LIN {X 0,Y 303.752,Z 774.326,A -85,B 0,C 180,E1 -15927.348,E2 -15927.348} C_VEL
LIN {X 0,Y 303.832,Z 775.153,A -85,B 0,C 180,E1 -15928.675,E2 -15928.675} C_VEL
LIN {X 0,Y 303.933,Z 775.529,A -85,B 0,C 180,E1 -15930,E2 -15930} C_VEL
LIN {X 0,Y 303.82,Z 775.489,A -85,B 0,C 180,E1 -15931.325,E2 -15931.325} C_VEL
LIN {X 0,Y 303.73,Z 775.052,A -85,B 0,C 180,E1 -15932.652,E2 -15932.652} C_VEL
LIN {X 0,Y 303.716,Z 774.21,A -85,B 0,C 180,E1 -15933.981,E2 -15933.981} C_VEL
LIN {X 0,Y 303.694,Z 772.494,A -85,B 0,C 180,E1 -15935.672,E2 -15935.672} C_VEL
LIN {X 0,Y 303.924,Z 769.081,A -85,B 0,C 180,E1 -15937.975,E2 -15937.975} C_VEL
LIN {X 0,Y 304.337,Z 764.982,A -85,B 0,C 180,E1 -15939.973,E2 -15939.973} C_VEL
LIN {X 0,Y 305.177,Z 758.726,A -85,B 0,C 180,E1 -15942.299,E2 -15942.299} C_VEL
LIN {X 0,Y 306.408,Z 751.923,A -85,B 0,C 180,E1 -15944.274,E2 -15944.274} C_VEL
LIN {X 0,Y 307.768,Z 744.025,A -85,B 0,C 180,E1 -15946.134,E2 -15946.134} C_VEL
LIN {X 0,Y 309.259,Z 734.984,A -85,B 0,C 180,E1 -15947.866,E2 -15947.866} C_VEL
LIN {X 0,Y 311.01,Z 724.473,A -85,B 0,C 180,E1 -15949.469,E2 -15949.469} C_VEL
LIN {X 0,Y 312.894,Z 712.7,A -85,B 0,C 180,E1 -15950.889,E2 -15950.889} C_VEL
LIN {X 0,Y 314.521,Z 701.015,A -85,B 0,C 180,E1 -15951.979,E2 -15951.979} C_VEL
LIN {X 0,Y 316.004,Z 687.738,A -85,B 0,C 180,E1 -15952.904,E2 -15952.904} C_VEL
LIN {X 0,Y 317.222,Z 674.465,A -85,B 0,C 180,E1 -15953.536,E2 -15953.536} C_VEL
LIN {X 0,Y 317.908,Z 658.285,A -85,B 0,C 180,E1 -15954.003,E2 -15954.003} C_VEL
LIN {X 0,Y 319.318,Z 607.887,A -85,B 0,C 180,E1 -15955.253,E2 -15955.253} C_VEL
LIN {X 0,Y 316.205,Z 584.31,A -85,B 0,C 180,E1 -15956.239,E2 -15956.239} C_VEL
LIN {X 0,Y 312.558,Z 565.353,A -85,B 0,C 180,E1 -15957.18,E2 -15957.18} C_VEL
LIN {X 0,Y 311.642,Z 560.399,A -85,B 0,C 180,E1 -15957.47,E2 -15957.47} C_VEL
LIN {X 0,Y 311.424,Z 557.383,A -85,B 0,C 180,E1 -15958.342,E2 -15958.342} C_VEL
LIN {X 0,Y 309.368,Z 547.286,A -85,B 0,C 180,E1 -15961.499,E2 -15961.499} C_VEL
LIN {X 0,Y 306.994,Z 537.185,A -85,B 0,C 180,E1 -15964.911,E2 -15964.911} C_VEL
LIN {X 0,Y 305.519,Z 531.43,A -85,B 0,C 180,E1 -15967.041,E2 -15967.041} C_VEL
LIN {X 0,Y 305.484,Z 531.431,A -85,B 0,C 180,E1 -15970.605,E2 -15970.605} C_VEL
LIN {X 0,Y 305.491,Z 531.432,A -85,B 0,C 180,E1 -15973.642,E2 -15973.642} C_VEL
LIN {X 0,Y 305.461,Z 531.431,A -85,B 0,C 180,E1 -15977.411,E2 -15977.411} C_VEL
LIN {X 0,Y 305.493,Z 531.431,A -85,B 0,C 180,E1 -15981.599,E2 -15981.599} C_VEL
LIN {X 0,Y 305.46,Z 531.435,A -85,B 0,C 180,E1 -15984.886,E2 -15984.886} C_VEL
LIN {X 0,Y 305.448,Z 531.435,A -85,B 0,C 180,E1 -15988.354,E2 -15988.354} C_VEL
LIN {X 0,Y 305.517,Z 531.428,A -85,B 0,C 180,E1 -15991.113,E2 -15991.113} C_VEL
LIN {X 0,Y 305.567,Z 531.422,A -85,B 0,C 180,E1 -15994.087,E2 -15994.087} C_VEL
LIN {X 0,Y 305.495,Z 531.429,A -85,B 0,C 180,E1 -15998.402,E2 -15998.402} C_VEL
LIN {X 0,Y 305.584,Z 531.42,A -85,B 0,C 180,E1 -16001.217,E2 -16001.217} C_VEL
LIN {X 0,Y 305.643,Z 531.411,A -85,B 0,C 180,E1 -16005.348,E2 -16005.348} C_VEL
LIN {X 0,Y 305.632,Z 531.409,A -85,B 0,C 180,E1 -16009.399,E2 -16009.399} C_VEL
LIN {X 0,Y 305.803,Z 531.392,A -85,B 0,C 180,E1 -16012.073,E2 -16012.073} C_VEL
LIN {X 0,Y 305.685,Z 531.404,A -85,B 0,C 180,E1 -16014.723,E2 -16014.723} C_VEL
LIN {X 0,Y 305.952,Z 531.374,A -85,B 0,C 180,E1 -16018.683,E2 -16018.683} C_VEL
LIN {X 0,Y 305.954,Z 531.373,A -85,B 0,C 180,E1 -16021.316,E2 -16021.316} C_VEL
LIN {X 0,Y 305.684,Z 531.408,A -85,B 0,C 180,E1 -16025.276,E2 -16025.276} C_VEL
LIN {X 0,Y 305.79,Z 531.394,A -85,B 0,C 180,E1 -16027.926,E2 -16027.926} C_VEL
LIN {X 0,Y 305.596,Z 531.418,A -85,B 0,C 180,E1 -16031.945,E2 -16031.945} C_VEL
LIN {X 0,Y 305.63,Z 531.417,A -85,B 0,C 180,E1 -16035.034,E2 -16035.034} C_VEL
LIN {X 0,Y 305.569,Z 531.422,A -85,B 0,C 180,E1 -16039.445,E2 -16039.445} C_VEL
LIN {X 0,Y 305.523,Z 531.521,A -85,B 0,C 180,E1 -16043.261,E2 -16043.261} C_VEL
LIN {X 0,Y 305.945,Z 533.184,A -85,B 0,C 180,E1 -16043.972,E2 -16043.972} C_VEL
LIN {X 0,Y 314.593,Z 550.365,A -85,B 0,C 180,E1 -16045.514,E2 -16045.514} C_VEL
LIN {X 0,Y 320.66,Z 564.718,A -85,B 0,C 180,E1 -16046.576,E2 -16046.576} C_VEL
LIN {X 0,Y 318.124,Z 639.345,A -85,B 0,C 180,E1 -16048.445,E2 -16048.445} C_VEL
LIN {X 0,Y 317.297,Z 653.008,A -85,B 0,C 180,E1 -16049.057,E2 -16049.057} C_VEL
LIN {X 0,Y 316.324,Z 664.988,A -85,B 0,C 180,E1 -16049.846,E2 -16049.846} C_VEL
LIN {X 0,Y 315.081,Z 676.532,A -85,B 0,C 180,E1 -16050.865,E2 -16050.865} C_VEL
LIN {X 0,Y 313.614,Z 687.468,A -85,B 0,C 180,E1 -16052.096,E2 -16052.096} C_VEL
LIN {X 0,Y 311.861,Z 698.493,A -85,B 0,C 180,E1 -16053.658,E2 -16053.658} C_VEL
LIN {X 0,Y 310.187,Z 707.916,A -85,B 0,C 180,E1 -16055.349,E2 -16055.349} C_VEL
LIN {X 0,Y 308.688,Z 716.087,A -85,B 0,C 180,E1 -16057.171,E2 -16057.171} C_VEL
LIN {X 0,Y 307.4,Z 722.671,A -85,B 0,C 180,E1 -16058.985,E2 -16058.985} C_VEL
LIN {X 0,Y 306.345,Z 727.975,A -85,B 0,C 180,E1 -16060.795,E2 -16060.795} C_VEL
LIN {X 0,Y 305.272,Z 733.419,A -85,B 0,C 180,E1 -16063.204,E2 -16063.204} C_VEL
LIN {X 0,Y 304.531,Z 737.329,A -85,B 0,C 180,E1 -16065.677,E2 -16065.677} C_VEL
LIN {X 0,Y 304.003,Z 739.571,A -85,B 0,C 180,E1 -16067.901,E2 -16067.901} C_VEL
LIN {X 0,Y 303.735,Z 740.546,A -85,B 0,C 180,E1 -16069.779,E2 -16069.779} C_VEL
LIN {X 0,Y 303.591,Z 740.689,A -85,B 0,C 180,E1 -16071.913,E2 -16071.913} C_VEL
LIN {X 0,Y 303.659,Z 739.758,A -85,B 0,C 180,E1 -16074.1,E2 -16074.1} C_VEL
LIN {X 0,Y 303.916,Z 737.644,A -85,B 0,C 180,E1 -16076.354,E2 -16076.354} C_VEL
LIN {X 0,Y 304.384,Z 734.163,A -85,B 0,C 180,E1 -16078.681,E2 -16078.681} C_VEL
LIN {X 0,Y 305.049,Z 728.962,A -85,B 0,C 180,E1 -16081.1,E2 -16081.1} C_VEL
LIN {X 0,Y 305.869,Z 723.125,A -85,B 0,C 180,E1 -16083.163,E2 -16083.163} C_VEL
LIN {X 0,Y 306.927,Z 715.425,A -85,B 0,C 180,E1 -16085.299,E2 -16085.299} C_VEL
LIN {X 0,Y 308.099,Z 706.856,A -85,B 0,C 180,E1 -16087.184,E2 -16087.184} C_VEL
LIN {X 0,Y 309.346,Z 697.634,A -85,B 0,C 180,E1 -16088.826,E2 -16088.826} C_VEL
LIN {X 0,Y 310.622,Z 687.259,A -85,B 0,C 180,E1 -16090.314,E2 -16090.314} C_VEL
LIN {X 0,Y 311.869,Z 675.857,A -85,B 0,C 180,E1 -16091.61,E2 -16091.61} C_VEL
LIN {X 0,Y 312.946,Z 663.701,A -85,B 0,C 180,E1 -16092.689,E2 -16092.689} C_VEL
LIN {X 0,Y 313.769,Z 651.237,A -85,B 0,C 180,E1 -16093.505,E2 -16093.505} C_VEL
LIN {X 0,Y 314.4,Z 638.134,A -85,B 0,C 180,E1 -16094.092,E2 -16094.092} C_VEL
LIN {X 0,Y 315.41,Z 601.901,A -85,B 0,C 180,E1 -16095.002,E2 -16095.002} C_VEL
LIN {X 0,Y 316.392,Z 560.015,A -85,B 0,C 180,E1 -16096.021,E2 -16096.021} C_VEL
LIN {X 0,Y 308.547,Z 538.734,A -85,B 0,C 180,E1 -16097.158,E2 -16097.158} C_VEL
LIN {X 0,Y 305.743,Z 532.085,A -85,B 0,C 180,E1 -16097.555,E2 -16097.555} C_VEL
LIN {X 0,Y 305.63,Z 531.415,A -85,B 0,C 180,E1 -16097.635,E2 -16097.635} C_VEL
LIN {X 0,Y 305.804,Z 531.392,A -85,B 0,C 180,E1 -16102.074,E2 -16102.074} C_VEL
LIN {X 0,Y 305.685,Z 531.409,A -85,B 0,C 180,E1 -16104.724,E2 -16104.724} C_VEL
LIN {X 0,Y 305.955,Z 531.375,A -85,B 0,C 180,E1 -16108.684,E2 -16108.684} C_VEL
LIN {X 0,Y 305.955,Z 531.373,A -85,B 0,C 180,E1 -16111.316,E2 -16111.316} C_VEL
LIN {X 0,Y 305.85,Z 531.387,A -85,B 0,C 180,E1 -16116.597,E2 -16116.597} C_VEL
LIN {X 0,Y 305.733,Z 531.401,A -85,B 0,C 180,E1 -16119.26,E2 -16119.26} C_VEL
LIN {X 0,Y 305.586,Z 531.419,A -85,B 0,C 180,E1 -16123.296,E2 -16123.296} C_VEL
LIN {X 0,Y 305.59,Z 531.416,A -85,B 0,C 180,E1 -16126.02,E2 -16126.02} C_VEL
LIN {X 0,Y 305.573,Z 531.419,A -85,B 0,C 180,E1 -16129.445,E2 -16129.445} C_VEL
LIN {X 0,Y 305.487,Z 531.434,A -85,B 0,C 180,E1 -16133.041,E2 -16133.041} C_VEL
LIN {X 0,Y 305.543,Z 531.422,A -85,B 0,C 180,E1 -16136.227,E2 -16136.227} C_VEL
LIN {X 0,Y 305.493,Z 531.433,A -85,B 0,C 180,E1 -16139.05,E2 -16139.05} C_VEL
LIN {X 0,Y 305.443,Z 531.435,A -85,B 0,C 180,E1 -16141.951,E2 -16141.951} C_VEL
LIN {X 0,Y 305.458,Z 531.438,A -85,B 0,C 180,E1 -16145.113,E2 -16145.113} C_VEL
LIN {X 0,Y 305.488,Z 531.429,A -85,B 0,C 180,E1 -16148.539,E2 -16148.539} C_VEL
LIN {X 0,Y 305.516,Z 531.427,A -85,B 0,C 180,E1 -16152.599,E2 -16152.599} C_VEL
LIN {X 0,Y 305.527,Z 531.423,A -85,B 0,C 180,E1 -16156.364,E2 -16156.364} C_VEL
LIN {X 0,Y 305.478,Z 531.429,A -85,B 0,C 180,E1 -16159.896,E2 -16159.896} C_VEL
LIN {X 0,Y 305.479,Z 531.432,A -85,B 0,C 180,E1 -16163.076,E2 -16163.076} C_VEL
LIN {X 0,Y 304.857,Z 531.517,A -85,B 0,C 180,E1 -16164.175,E2 -16164.175} C_VEL
LIN {X 0,Y 302.011,Z 531.875,A -85,B 0,C 180,E1 -16165.964,E2 -16165.964} C_VEL
LIN {X 0,Y 299.555,Z 532.175,A -85,B 0,C 180,E1 -16167.416,E2 -16167.416} C_VEL
LIN {X 0,Y 298.479,Z 532.302,A -85,B 0,C 180,E1 -16168.54,E2 -16168.54} C_VEL
LIN {X 0,Y 298.381,Z 532.311,A -85,B 0,C 180,E1 -16168.922,E2 -16168.922} C_VEL
LIN {X 0,Y 298.462,Z 532.304,A -85,B 0,C 180,E1 -16171.905,E2 -16171.905} C_VEL
LIN {X 0,Y 298.477,Z 532.306,A -85,B 0,C 180,E1 -16174.924,E2 -16174.924} C_VEL
LIN {X 0,Y 298.429,Z 532.309,A -85,B 0,C 180,E1 -16179.315,E2 -16179.315} C_VEL
LIN {X 0,Y 298.527,Z 532.295,A -85,B 0,C 180,E1 -16182.179,E2 -16182.179} C_VEL
LIN {X 0,Y 298.586,Z 532.292,A -85,B 0,C 180,E1 -16184.995,E2 -16184.995} C_VEL
LIN {X 0,Y 298.588,Z 532.289,A -85,B 0,C 180,E1 -16189.147,E2 -16189.147} C_VEL
LIN {X 0,Y 298.752,Z 532.266,A -85,B 0,C 180,E1 -16191.886,E2 -16191.886} C_VEL
LIN {X 0,Y 298.657,Z 532.28,A -85,B 0,C 180,E1 -16194.6,E2 -16194.6} C_VEL
LIN {X 0,Y 298.918,Z 532.247,A -85,B 0,C 180,E1 -16198.653,E2 -16198.653} C_VEL
LIN {X 0,Y 298.922,Z 532.249,A -85,B 0,C 180,E1 -16201.348,E2 -16201.348} C_VEL
LIN {X 0,Y 298.657,Z 532.283,A -85,B 0,C 180,E1 -16205.402,E2 -16205.402} C_VEL
LIN {X 0,Y 298.735,Z 532.268,A -85,B 0,C 180,E1 -16208.115,E2 -16208.115} C_VEL
LIN {X 0,Y 298.547,Z 532.293,A -85,B 0,C 180,E1 -16212.232,E2 -16212.232} C_VEL
LIN {X 0,Y 298.601,Z 532.292,A -85,B 0,C 180,E1 -16215.21,E2 -16215.21} C_VEL
LIN {X 0,Y 298.534,Z 532.299,A -85,B 0,C 180,E1 -16219.244,E2 -16219.244} C_VEL
LIN {X 0,Y 298.453,Z 532.306,A -85,B 0,C 180,E1 -16223.599,E2 -16223.599} C_VEL
LIN {X 0,Y 298.486,Z 532.302,A -85,B 0,C 180,E1 -16226.575,E2 -16226.575} C_VEL
LIN {X 0,Y 298.418,Z 532.312,A -85,B 0,C 180,E1 -16229.642,E2 -16229.642} C_VEL
LIN {X 0,Y 298.394,Z 532.314,A -85,B 0,C 180,E1 -16232.801,E2 -16232.801} C_VEL
LIN {X 0,Y 298.462,Z 532.306,A -85,B 0,C 180,E1 -16236.813,E2 -16236.813} C_VEL
LIN {X 0,Y 298.386,Z 532.317,A -85,B 0,C 180,E1 -16241.089,E2 -16241.089} C_VEL
LIN {X 0,Y 298.416,Z 532.313,A -85,B 0,C 180,E1 -16244.954,E2 -16244.954} C_VEL
LIN {X 0,Y 298.451,Z 532.307,A -85,B 0,C 180,E1 -16248.751,E2 -16248.751} C_VEL
LIN {X 0,Y 298.47,Z 532.308,A -85,B 0,C 180,E1 -16253.187,E2 -16253.187} C_VEL
LIN {X 0,Y 298.45,Z 532.331,A -85,B 0,C 180,E1 -16255.348,E2 -16255.348} C_VEL
LIN {X 0,Y 301.104,Z 544.622,A -85,B 0,C 180,E1 -16259.104,E2 -16259.104} C_VEL
LIN {X 0,Y 303.404,Z 555.956,A -85,B 0,C 180,E1 -16262.402,E2 -16262.402} C_VEL
LIN {X 0,Y 303.106,Z 560.058,A -85,B 0,C 180,E1 -16263.491,E2 -16263.491} C_VEL
LIN {X 0,Y 302.801,Z 562.624,A -85,B 0,C 180,E1 -16264.161,E2 -16264.161} C_VEL
LIN {X 0,Y 308.8,Z 606.859,A -85,B 0,C 180,E1 -16265.801,E2 -16265.801} C_VEL
LIN {X 0,Y 308.7,Z 621.69,A -85,B 0,C 180,E1 -16266.186,E2 -16266.186} C_VEL
LIN {X 0,Y 307.289,Z 672.374,A -85,B 0,C 180,E1 -16267.475,E2 -16267.475} C_VEL
LIN {X 0,Y 306.417,Z 685.767,A -85,B 0,C 180,E1 -16268.073,E2 -16268.073} C_VEL
LIN {X 0,Y 305.187,Z 698.528,A -85,B 0,C 180,E1 -16268.911,E2 -16268.911} C_VEL
LIN {X 0,Y 303.826,Z 711.076,A -85,B 0,C 180,E1 -16270.051,E2 -16270.051} C_VEL
LIN {X 0,Y 302.31,Z 722.294,A -85,B 0,C 180,E1 -16271.358,E2 -16271.358} C_VEL
LIN {X 0,Y 301.15,Z 731.415,A -85,B 0,C 180,E1 -16272.69,E2 -16272.69} C_VEL
LIN {X 0,Y 299.917,Z 740.863,A -85,B 0,C 180,E1 -16274.388,E2 -16274.388} C_VEL
LIN {X 0,Y 298.705,Z 749.842,A -85,B 0,C 180,E1 -16276.392,E2 -16276.392} C_VEL
LIN {X 0,Y 297.668,Z 757.125,A -85,B 0,C 180,E1 -16278.423,E2 -16278.423} C_VEL
LIN {X 0,Y 297.117,Z 762.927,A -85,B 0,C 180,E1 -16280.469,E2 -16280.469} C_VEL
LIN {X 0,Y 296.795,Z 767.473,A -85,B 0,C 180,E1 -16282.517,E2 -16282.517} C_VEL
LIN {X 0,Y 296.671,Z 770.897,A -85,B 0,C 180,E1 -16284.563,E2 -16284.563} C_VEL
LIN {X 0,Y 296.687,Z 772.586,A -85,B 0,C 180,E1 -16285.925,E2 -16285.925} C_VEL
LIN {X 0,Y 296.673,Z 773.85,A -85,B 0,C 180,E1 -16287.284,E2 -16287.284} C_VEL
LIN {X 0,Y 296.739,Z 774.705,A -85,B 0,C 180,E1 -16288.643,E2 -16288.643} C_VEL
LIN {X 0,Y 296.844,Z 775.107,A -85,B 0,C 180,E1 -16290,E2 -16290} C_VEL
LIN {X 0,Y 296.725,Z 775.084,A -85,B 0,C 180,E1 -16291.357,E2 -16291.357} C_VEL
LIN {X 0,Y 296.649,Z 774.665,A -85,B 0,C 180,E1 -16292.716,E2 -16292.716} C_VEL
LIN {X 0,Y 296.627,Z 773.847,A -85,B 0,C 180,E1 -16294.076,E2 -16294.076} C_VEL
LIN {X 0,Y 296.608,Z 772.362,A -85,B 0,C 180,E1 -16295.626,E2 -16295.626} C_VEL
LIN {X 0,Y 296.86,Z 768.775,A -85,B 0,C 180,E1 -16298.166,E2 -16298.166} C_VEL
LIN {X 0,Y 297.324,Z 764.721,A -85,B 0,C 180,E1 -16300.211,E2 -16300.211} C_VEL
LIN {X 0,Y 298.21,Z 758.544,A -85,B 0,C 180,E1 -16302.591,E2 -16302.591} C_VEL
LIN {X 0,Y 299.492,Z 751.806,A -85,B 0,C 180,E1 -16304.611,E2 -16304.611} C_VEL
LIN {X 0,Y 300.99,Z 743.534,A -85,B 0,C 180,E1 -16306.606,E2 -16306.606} C_VEL
LIN {X 0,Y 302.486,Z 734.997,A -85,B 0,C 180,E1 -16308.28,E2 -16308.28} C_VEL
LIN {X 0,Y 304.347,Z 724.612,A -85,B 0,C 180,E1 -16309.913,E2 -16309.913} C_VEL
LIN {X 0,Y 306.292,Z 712.956,A -85,B 0,C 180,E1 -16311.361,E2 -16311.361} C_VEL
LIN {X 0,Y 307.968,Z 701.517,A -85,B 0,C 180,E1 -16312.472,E2 -16312.472} C_VEL
LIN {X 0,Y 309.514,Z 688.59,A -85,B 0,C 180,E1 -16313.413,E2 -16313.413} C_VEL
LIN {X 0,Y 310.838,Z 675.214,A -85,B 0,C 180,E1 -16314.089,E2 -16314.089} C_VEL
LIN {X 0,Y 311.593,Z 660.428,A -85,B 0,C 180,E1 -16314.547,E2 -16314.547} C_VEL
LIN {X 0,Y 313.156,Z 609.092,A -85,B 0,C 180,E1 -16315.847,E2 -16315.847} C_VEL
LIN {X 0,Y 310.081,Z 585.474,A -85,B 0,C 180,E1 -16316.864,E2 -16316.864} C_VEL
LIN {X 0,Y 305.766,Z 563.081,A -85,B 0,C 180,E1 -16318.032,E2 -16318.032} C_VEL
LIN {X 0,Y 304.741,Z 559.888,A -85,B 0,C 180,E1 -16318.295,E2 -16318.295} C_VEL
LIN {X 0,Y 302.745,Z 549.914,A -85,B 0,C 180,E1 -16321.486,E2 -16321.486} C_VEL
LIN {X 0,Y 300.622,Z 540.588,A -85,B 0,C 180,E1 -16324.7,E2 -16324.7} C_VEL
LIN {X 0,Y 298.485,Z 532.306,A -85,B 0,C 180,E1 -16327.853,E2 -16327.853} C_VEL
LIN {X 0,Y 298.451,Z 532.307,A -85,B 0,C 180,E1 -16331.249,E2 -16331.249} C_VEL
LIN {X 0,Y 298.416,Z 532.31,A -85,B 0,C 180,E1 -16335.046,E2 -16335.046} C_VEL
LIN {X 0,Y 298.387,Z 532.319,A -85,B 0,C 180,E1 -16338.911,E2 -16338.911} C_VEL
LIN {X 0,Y 298.462,Z 532.303,A -85,B 0,C 180,E1 -16343.187,E2 -16343.187} C_VEL
LIN {X 0,Y 298.392,Z 532.317,A -85,B 0,C 180,E1 -16347.199,E2 -16347.199} C_VEL
LIN {X 0,Y 298.428,Z 532.312,A -85,B 0,C 180,E1 -16350.614,E2 -16350.614} C_VEL
LIN {X 0,Y 298.48,Z 532.305,A -85,B 0,C 180,E1 -16353.473,E2 -16353.473} C_VEL
LIN {X 0,Y 298.43,Z 532.307,A -85,B 0,C 180,E1 -16356.697,E2 -16356.697} C_VEL
LIN {X 0,Y 298.534,Z 532.298,A -85,B 0,C 180,E1 -16360.756,E2 -16360.756} C_VEL
LIN {X 0,Y 298.588,Z 532.292,A -85,B 0,C 180,E1 -16364.994,E2 -16364.994} C_VEL
LIN {X 0,Y 298.587,Z 532.288,A -85,B 0,C 180,E1 -16369.146,E2 -16369.146} C_VEL
LIN {X 0,Y 298.749,Z 532.271,A -85,B 0,C 180,E1 -16371.885,E2 -16371.885} C_VEL
LIN {X 0,Y 298.655,Z 532.278,A -85,B 0,C 180,E1 -16374.598,E2 -16374.598} C_VEL
LIN {X 0,Y 298.918,Z 532.25,A -85,B 0,C 180,E1 -16378.652,E2 -16378.652} C_VEL
LIN {X 0,Y 298.92,Z 532.249,A -85,B 0,C 180,E1 -16381.347,E2 -16381.347} C_VEL
LIN {X 0,Y 298.654,Z 532.283,A -85,B 0,C 180,E1 -16385.401,E2 -16385.401} C_VEL
LIN {X 0,Y 298.735,Z 532.273,A -85,B 0,C 180,E1 -16388.114,E2 -16388.114} C_VEL
LIN {X 0,Y 298.546,Z 532.297,A -85,B 0,C 180,E1 -16392.231,E2 -16392.231} C_VEL
LIN {X 0,Y 298.578,Z 532.294,A -85,B 0,C 180,E1 -16395.194,E2 -16395.194} C_VEL
LIN {X 0,Y 298.532,Z 532.298,A -85,B 0,C 180,E1 -16399.243,E2 -16399.243} C_VEL
LIN {X 0,Y 298.487,Z 532.483,A -85,B 0,C 180,E1 -16402.519,E2 -16402.519} C_VEL
LIN {X 0,Y 298.802,Z 533.739,A -85,B 0,C 180,E1 -16403.078,E2 -16403.078} C_VEL
LIN {X 0,Y 306.903,Z 549.266,A -85,B 0,C 180,E1 -16404.591,E2 -16404.591} C_VEL
LIN {X 0,Y 312.984,Z 562.829,A -85,B 0,C 180,E1 -16405.699,E2 -16405.699} C_VEL
LIN {X 0,Y 314.495,Z 567.114,A -85,B 0,C 180,E1 -16405.989,E2 -16405.989} C_VEL
LIN {X 0,Y 311.879,Z 639.717,A -85,B 0,C 180,E1 -16407.841,E2 -16407.841} C_VEL
LIN {X 0,Y 310.992,Z 653.473,A -85,B 0,C 180,E1 -16408.469,E2 -16408.469} C_VEL
LIN {X 0,Y 309.858,Z 666.611,A -85,B 0,C 180,E1 -16409.372,E2 -16409.372} C_VEL
LIN {X 0,Y 308.314,Z 679.449,A -85,B 0,C 180,E1 -16410.57,E2 -16410.57} C_VEL
LIN {X 0,Y 306.624,Z 691.13,A -85,B 0,C 180,E1 -16412.001,E2 -16412.001} C_VEL
LIN {X 0,Y 304.847,Z 701.437,A -85,B 0,C 180,E1 -16413.593,E2 -16413.593} C_VEL
LIN {X 0,Y 303.015,Z 710.983,A -85,B 0,C 180,E1 -16415.438,E2 -16415.438} C_VEL
LIN {X 0,Y 301.332,Z 719.489,A -85,B 0,C 180,E1 -16417.536,E2 -16417.536} C_VEL
LIN {X 0,Y 300.051,Z 725.487,A -85,B 0,C 180,E1 -16419.382,E2 -16419.382} C_VEL
LIN {X 0,Y 298.844,Z 731.397,A -85,B 0,C 180,E1 -16421.699,E2 -16421.699} C_VEL
LIN {X 0,Y 297.946,Z 735.735,A -85,B 0,C 180,E1 -16424.012,E2 -16424.012} C_VEL
LIN {X 0,Y 297.601,Z 737.326,A -85,B 0,C 180,E1 -16425.109,E2 -16425.109} C_VEL
LIN {X 0,Y 297.061,Z 739.557,A -85,B 0,C 180,E1 -16427.172,E2 -16427.172} C_VEL
LIN {X 0,Y 296.713,Z 740.85,A -85,B 0,C 180,E1 -16429.283,E2 -16429.283} C_VEL
LIN {X 0,Y 296.518,Z 741.083,A -85,B 0,C 180,E1 -16431.959,E2 -16431.959} C_VEL
LIN {X 0,Y 296.549,Z 740.416,A -85,B 0,C 180,E1 -16433.684,E2 -16433.684} C_VEL
LIN {X 0,Y 296.759,Z 738.496,A -85,B 0,C 180,E1 -16435.983,E2 -16435.983} C_VEL
LIN {X 0,Y 297.31,Z 734.739,A -85,B 0,C 180,E1 -16438.665,E2 -16438.665} C_VEL
LIN {X 0,Y 297.854,Z 730.399,A -85,B 0,C 180,E1 -16440.811,E2 -16440.811} C_VEL
LIN {X 0,Y 298.712,Z 724.404,A -85,B 0,C 180,E1 -16443.058,E2 -16443.058} C_VEL
LIN {X 0,Y 299.654,Z 717.755,A -85,B 0,C 180,E1 -16445.029,E2 -16445.029} C_VEL
LIN {X 0,Y 300.832,Z 709.654,A -85,B 0,C 180,E1 -16446.965,E2 -16446.965} C_VEL
LIN {X 0,Y 302.071,Z 700.698,A -85,B 0,C 180,E1 -16448.686,E2 -16448.686} C_VEL
LIN {X 0,Y 303.526,Z 689.674,A -85,B 0,C 180,E1 -16450.383,E2 -16450.383} C_VEL
LIN {X 0,Y 304.748,Z 679.065,A -85,B 0,C 180,E1 -16451.687,E2 -16451.687} C_VEL
LIN {X 0,Y 305.859,Z 667.604,A -85,B 0,C 180,E1 -16452.793,E2 -16452.793} C_VEL
LIN {X 0,Y 306.883,Z 654.523,A -85,B 0,C 180,E1 -16453.742,E2 -16453.742} C_VEL
LIN {X 0,Y 307.58,Z 642.289,A -85,B 0,C 180,E1 -16454.37,E2 -16454.37} C_VEL
LIN {X 0,Y 308.082,Z 627.719,A -85,B 0,C 180,E1 -16454.819,E2 -16454.819} C_VEL
LIN {X 0,Y 309.827,Z 561.637,A -85,B 0,C 180,E1 -16456.448,E2 -16456.448} C_VEL
LIN {X 0,Y 302.536,Z 541.906,A -85,B 0,C 180,E1 -16457.534,E2 -16457.534} C_VEL
LIN {X 0,Y 298.733,Z 533.084,A -85,B 0,C 180,E1 -16458.078,E2 -16458.078} C_VEL
LIN {X 0,Y 298.588,Z 532.293,A -85,B 0,C 180,E1 -16458.115,E2 -16458.115} C_VEL
LIN {X 0,Y 298.75,Z 532.271,A -85,B 0,C 180,E1 -16461.886,E2 -16461.886} C_VEL
LIN {X 0,Y 298.655,Z 532.284,A -85,B 0,C 180,E1 -16464.599,E2 -16464.599} C_VEL
LIN {X 0,Y 298.921,Z 532.251,A -85,B 0,C 180,E1 -16468.653,E2 -16468.653} C_VEL
LIN {X 0,Y 298.921,Z 532.25,A -85,B 0,C 180,E1 -16471.347,E2 -16471.347} C_VEL
LIN {X 0,Y 298.795,Z 532.267,A -85,B 0,C 180,E1 -16476.754,E2 -16476.754} C_VEL
LIN {X 0,Y 298.677,Z 532.279,A -85,B 0,C 180,E1 -16479.48,E2 -16479.48} C_VEL
LIN {X 0,Y 298.549,Z 532.293,A -85,B 0,C 180,E1 -16483.615,E2 -16483.615} C_VEL
LIN {X 0,Y 298.545,Z 532.294,A -85,B 0,C 180,E1 -16486.408,E2 -16486.408} C_VEL
LIN {X 0,Y 298.508,Z 532.298,A -85,B 0,C 180,E1 -16489.655,E2 -16489.655} C_VEL
LIN {X 0,Y 298.453,Z 532.306,A -85,B 0,C 180,E1 -16493.597,E2 -16493.597} C_VEL
LIN {X 0,Y 298.485,Z 532.302,A -85,B 0,C 180,E1 -16496.574,E2 -16496.574} C_VEL
LIN {X 0,Y 298.418,Z 532.31,A -85,B 0,C 180,E1 -16499.64,E2 -16499.64} C_VEL
LIN {X 0,Y 298.393,Z 532.316,A -85,B 0,C 180,E1 -16502.8,E2 -16502.8} C_VEL
LIN {X 0,Y 298.465,Z 532.307,A -85,B 0,C 180,E1 -16506.814,E2 -16506.814} C_VEL
LIN {X 0,Y 298.451,Z 532.309,A -85,B 0,C 180,E1 -16511.249,E2 -16511.249} C_VEL
LIN {X 0,Y 298.483,Z 532.306,A -85,B 0,C 180,E1 -16515.061,E2 -16515.061} C_VEL
LIN {X 0,Y 298.447,Z 532.306,A -85,B 0,C 180,E1 -16518.898,E2 -16518.898} C_VEL
LIN {X 0,Y 298.459,Z 532.309,A -85,B 0,C 180,E1 -16523.187,E2 -16523.187} C_VEL
LIN {X 0,Y 298.388,Z 532.313,A -85,B 0,C 180,E1 -16527.2,E2 -16527.2} C_VEL
LIN {X 0,Y 298.381,Z 532.311,A -85,B 0,C 180,E1 -16528.922,E2 -16528.922} C_VEL
LIN {X 0,Y 297.698,Z 532.398,A -85,B 0,C 180,E1 -16530.05,E2 -16530.05} C_VEL
LIN {X 0,Y 294.88,Z 532.75,A -85,B 0,C 180,E1 -16531.888,E2 -16531.888} C_VEL
LIN {X 0,Y 292.497,Z 533.05,A -85,B 0,C 180,E1 -16533.379,E2 -16533.379} C_VEL
LIN {X 0,Y 291.462,Z 533.177,A -85,B 0,C 180,E1 -16534.533,E2 -16534.533} C_VEL
LIN {X 0,Y 291.371,Z 533.184,A -85,B 0,C 180,E1 -16534.924,E2 -16534.924} C_VEL
LIN {X 0,Y 291.356,Z 533.188,A -85,B 0,C 180,E1 -16538.788,E2 -16538.788} C_VEL
LIN {X 0,Y 291.46,Z 533.176,A -85,B 0,C 180,E1 -16541.732,E2 -16541.732} C_VEL
LIN {X 0,Y 291.533,Z 533.168,A -85,B 0,C 180,E1 -16544.635,E2 -16544.635} C_VEL
LIN {X 0,Y 291.531,Z 533.168,A -85,B 0,C 180,E1 -16548.881,E2 -16548.881} C_VEL
LIN {X 0,Y 291.702,Z 533.144,A -85,B 0,C 180,E1 -16551.689,E2 -16551.689} C_VEL
LIN {X 0,Y 291.627,Z 533.155,A -85,B 0,C 180,E1 -16554.469,E2 -16554.469} C_VEL
LIN {X 0,Y 291.884,Z 533.122,A -85,B 0,C 180,E1 -16558.621,E2 -16558.621} C_VEL
LIN {X 0,Y 291.889,Z 533.124,A -85,B 0,C 180,E1 -16561.38,E2 -16561.38} C_VEL
LIN {X 0,Y 291.626,Z 533.158,A -85,B 0,C 180,E1 -16565.532,E2 -16565.532} C_VEL
LIN {X 0,Y 291.682,Z 533.146,A -85,B 0,C 180,E1 -16568.313,E2 -16568.313} C_VEL
LIN {X 0,Y 291.514,Z 533.17,A -85,B 0,C 180,E1 -16572.532,E2 -16572.532} C_VEL
LIN {X 0,Y 291.55,Z 533.168,A -85,B 0,C 180,E1 -16575.377,E2 -16575.377} C_VEL
LIN {X 0,Y 291.446,Z 533.179,A -85,B 0,C 180,E1 -16579.876,E2 -16579.876} C_VEL
LIN {X 0,Y 291.396,Z 533.183,A -85,B 0,C 180,E1 -16584.206,E2 -16584.206} C_VEL
LIN {X 0,Y 291.419,Z 533.187,A -85,B 0,C 180,E1 -16587.273,E2 -16587.273} C_VEL
LIN {X 0,Y 291.336,Z 533.192,A -85,B 0,C 180,E1 -16590.438,E2 -16590.438} C_VEL
LIN {X 0,Y 291.343,Z 533.193,A -85,B 0,C 180,E1 -16593.699,E2 -16593.699} C_VEL
LIN {X 0,Y 291.387,Z 533.19,A -85,B 0,C 180,E1 -16597.258,E2 -16597.258} C_VEL
LIN {X 0,Y 291.332,Z 533.193,A -85,B 0,C 180,E1 -16600.644,E2 -16600.644} C_VEL
LIN {X 0,Y 291.341,Z 533.192,A -85,B 0,C 180,E1 -16604.393,E2 -16604.393} C_VEL
LIN {X 0,Y 291.386,Z 533.187,A -85,B 0,C 180,E1 -16608.392,E2 -16608.392} C_VEL
LIN {X 0,Y 291.385,Z 533.191,A -85,B 0,C 180,E1 -16611.165,E2 -16611.165} C_VEL
LIN {X 0,Y 291.411,Z 533.247,A -85,B 0,C 180,E1 -16614.919,E2 -16614.919} C_VEL
LIN {X 0,Y 294.142,Z 545.801,A -85,B 0,C 180,E1 -16618.862,E2 -16618.862} C_VEL
LIN {X 0,Y 296.305,Z 556.539,A -85,B 0,C 180,E1 -16622.067,E2 -16622.067} C_VEL
LIN {X 0,Y 296.424,Z 559.312,A -85,B 0,C 180,E1 -16622.845,E2 -16622.845} C_VEL
LIN {X 0,Y 296.027,Z 562.183,A -85,B 0,C 180,E1 -16623.61,E2 -16623.61} C_VEL
LIN {X 0,Y 301.815,Z 604.82,A -85,B 0,C 180,E1 -16625.252,E2 -16625.252} C_VEL
LIN {X 0,Y 302.31,Z 610.604,A -85,B 0,C 180,E1 -16625.445,E2 -16625.445} C_VEL
LIN {X 0,Y 300.603,Z 671.977,A -85,B 0,C 180,E1 -16627.037,E2 -16627.037} C_VEL
LIN {X 0,Y 299.682,Z 685.355,A -85,B 0,C 180,E1 -16627.645,E2 -16627.645} C_VEL
LIN {X 0,Y 298.429,Z 698.122,A -85,B 0,C 180,E1 -16628.501,E2 -16628.501} C_VEL
LIN {X 0,Y 297.121,Z 709.877,A -85,B 0,C 180,E1 -16629.581,E2 -16629.581} C_VEL
LIN {X 0,Y 295.598,Z 721.247,A -85,B 0,C 180,E1 -16630.919,E2 -16630.919} C_VEL
LIN {X 0,Y 294.182,Z 731.522,A -85,B 0,C 180,E1 -16632.446,E2 -16632.446} C_VEL
LIN {X 0,Y 292.95,Z 740.503,A -85,B 0,C 180,E1 -16634.105,E2 -16634.105} C_VEL
LIN {X 0,Y 291.739,Z 749.096,A -85,B 0,C 180,E1 -16636.061,E2 -16636.061} C_VEL
LIN {X 0,Y 290.683,Z 756.448,A -85,B 0,C 180,E1 -16638.141,E2 -16638.141} C_VEL
LIN {X 0,Y 290.082,Z 762.32,A -85,B 0,C 180,E1 -16640.236,E2 -16640.236} C_VEL
LIN {X 0,Y 289.72,Z 766.913,A -85,B 0,C 180,E1 -16642.333,E2 -16642.333} C_VEL
LIN {X 0,Y 289.607,Z 770.382,A -85,B 0,C 180,E1 -16644.43,E2 -16644.43} C_VEL
LIN {X 0,Y 289.599,Z 772.09,A -85,B 0,C 180,E1 -16645.825,E2 -16645.825} C_VEL
LIN {X 0,Y 289.595,Z 773.374,A -85,B 0,C 180,E1 -16647.218,E2 -16647.218} C_VEL
LIN {X 0,Y 289.647,Z 774.251,A -85,B 0,C 180,E1 -16648.61,E2 -16648.61} C_VEL
LIN {X 0,Y 289.754,Z 774.686,A -85,B 0,C 180,E1 -16650,E2 -16650} C_VEL
LIN {X 0,Y 289.633,Z 774.68,A -85,B 0,C 180,E1 -16651.39,E2 -16651.39} C_VEL
LIN {X 0,Y 289.57,Z 774.278,A -85,B 0,C 180,E1 -16652.782,E2 -16652.782} C_VEL
LIN {X 0,Y 289.54,Z 773.481,A -85,B 0,C 180,E1 -16654.176,E2 -16654.176} C_VEL
LIN {X 0,Y 289.519,Z 772.247,A -85,B 0,C 180,E1 -16655.572,E2 -16655.572} C_VEL
LIN {X 0,Y 289.705,Z 769.613,A -85,B 0,C 180,E1 -16657.667,E2 -16657.667} C_VEL
LIN {X 0,Y 290.089,Z 765.959,A -85,B 0,C 180,E1 -16659.764,E2 -16659.764} C_VEL
LIN {X 0,Y 290.748,Z 761.204,A -85,B 0,C 180,E1 -16661.856,E2 -16661.856} C_VEL
LIN {X 0,Y 292.144,Z 754.067,A -85,B 0,C 180,E1 -16664.275,E2 -16664.275} C_VEL
LIN {X 0,Y 293.642,Z 746.383,A -85,B 0,C 180,E1 -16666.333,E2 -16666.333} C_VEL
LIN {X 0,Y 295.064,Z 738.577,A -85,B 0,C 180,E1 -16668.037,E2 -16668.037} C_VEL
LIN {X 0,Y 297.07,Z 728.075,A -85,B 0,C 180,E1 -16669.881,E2 -16669.881} C_VEL
LIN {X 0,Y 299.01,Z 717.438,A -85,B 0,C 180,E1 -16671.365,E2 -16671.365} C_VEL
LIN {X 0,Y 300.943,Z 705.611,A -85,B 0,C 180,E1 -16672.664,E2 -16672.664} C_VEL
LIN {X 0,Y 302.632,Z 693.074,A -85,B 0,C 180,E1 -16673.706,E2 -16673.706} C_VEL
LIN {X 0,Y 304.142,Z 679.993,A -85,B 0,C 180,E1 -16674.487,E2 -16674.487} C_VEL
LIN {X 0,Y 305.14,Z 666.363,A -85,B 0,C 180,E1 -16675.013,E2 -16675.013} C_VEL
LIN {X 0,Y 306.976,Z 609.841,A -85,B 0,C 180,E1 -16676.485,E2 -16676.485} C_VEL
LIN {X 0,Y 304.005,Z 586.779,A -85,B 0,C 180,E1 -16677.517,E2 -16677.517} C_VEL
LIN {X 0,Y 300.27,Z 566.853,A -85,B 0,C 180,E1 -16678.588,E2 -16678.588} C_VEL
LIN {X 0,Y 298.814,Z 562.696,A -85,B 0,C 180,E1 -16678.902,E2 -16678.902} C_VEL
LIN {X 0,Y 297.521,Z 559.357,A -85,B 0,C 180,E1 -16679.222,E2 -16679.222} C_VEL
LIN {X 0,Y 295.609,Z 550.042,A -85,B 0,C 180,E1 -16682.338,E2 -16682.338} C_VEL
LIN {X 0,Y 293.536,Z 541.255,A -85,B 0,C 180,E1 -16685.506,E2 -16685.506} C_VEL
LIN {X 0,Y 291.411,Z 533.185,A -85,B 0,C 180,E1 -16688.733,E2 -16688.733} C_VEL
LIN {X 0,Y 291.398,Z 533.186,A -85,B 0,C 180,E1 -16692.477,E2 -16692.477} C_VEL
LIN {X 0,Y 291.346,Z 533.195,A -85,B 0,C 180,E1 -16696.357,E2 -16696.357} C_VEL
LIN {X 0,Y 291.385,Z 533.184,A -85,B 0,C 180,E1 -16700.516,E2 -16700.516} C_VEL
LIN {X 0,Y 291.422,Z 533.179,A -85,B 0,C 180,E1 -16702.921,E2 -16702.921} C_VEL
LIN {X 0,Y 291.342,Z 533.188,A -85,B 0,C 180,E1 -16706.301,E2 -16706.301} C_VEL
LIN {X 0,Y 291.384,Z 533.188,A -85,B 0,C 180,E1 -16710.259,E2 -16710.259} C_VEL
LIN {X 0,Y 291.413,Z 533.186,A -85,B 0,C 180,E1 -16714.271,E2 -16714.271} C_VEL
LIN {X 0,Y 291.376,Z 533.191,A -85,B 0,C 180,E1 -16717.298,E2 -16717.298} C_VEL
LIN {X 0,Y 291.453,Z 533.177,A -85,B 0,C 180,E1 -16720.269,E2 -16720.269} C_VEL
LIN {X 0,Y 291.55,Z 533.169,A -85,B 0,C 180,E1 -16724.623,E2 -16724.623} C_VEL
LIN {X 0,Y 291.531,Z 533.17,A -85,B 0,C 180,E1 -16728.88,E2 -16728.88} C_VEL
LIN {X 0,Y 291.701,Z 533.149,A -85,B 0,C 180,E1 -16731.688,E2 -16731.688} C_VEL
LIN {X 0,Y 291.625,Z 533.153,A -85,B 0,C 180,E1 -16734.468,E2 -16734.468} C_VEL
LIN {X 0,Y 291.884,Z 533.126,A -85,B 0,C 180,E1 -16738.62,E2 -16738.62} C_VEL
LIN {X 0,Y 291.887,Z 533.125,A -85,B 0,C 180,E1 -16741.379,E2 -16741.379} C_VEL
LIN {X 0,Y 291.698,Z 533.145,A -85,B 0,C 180,E1 -16746.662,E2 -16746.662} C_VEL
LIN {X 0,Y 291.568,Z 533.166,A -85,B 0,C 180,E1 -16749.713,E2 -16749.713} C_VEL
LIN {X 0,Y 291.514,Z 533.172,A -85,B 0,C 180,E1 -16753.95,E2 -16753.95} C_VEL
LIN {X 0,Y 291.48,Z 533.18,A -85,B 0,C 180,E1 -16756.818,E2 -16756.818} C_VEL
LIN {X 0,Y 291.444,Z 533.183,A -85,B 0,C 180,E1 -16759.875,E2 -16759.875} C_VEL
LIN {X 0,Y 291.392,Z 533.361,A -85,B 0,C 180,E1 -16761.673,E2 -16761.673} C_VEL
LIN {X 0,Y 291.676,Z 534.477,A -85,B 0,C 180,E1 -16762.116,E2 -16762.116} C_VEL
LIN {X 0,Y 299.644,Z 549.057,A -85,B 0,C 180,E1 -16763.681,E2 -16763.681} C_VEL
LIN {X 0,Y 306.716,Z 564.314,A -85,B 0,C 180,E1 -16765.027,E2 -16765.027} C_VEL
LIN {X 0,Y 308.341,Z 568.662,A -85,B 0,C 180,E1 -16765.35,E2 -16765.35} C_VEL
LIN {X 0,Y 305.672,Z 640.138,A -85,B 0,C 180,E1 -16767.214,E2 -16767.214} C_VEL
LIN {X 0,Y 304.73,Z 653.741,A -85,B 0,C 180,E1 -16767.842,E2 -16767.842} C_VEL
LIN {X 0,Y 303.636,Z 666.238,A -85,B 0,C 180,E1 -16768.703,E2 -16768.703} C_VEL
LIN {X 0,Y 302.207,Z 678.096,A -85,B 0,C 180,E1 -16769.805,E2 -16769.805} C_VEL
LIN {X 0,Y 300.497,Z 689.488,A -85,B 0,C 180,E1 -16771.161,E2 -16771.161} C_VEL
LIN {X 0,Y 298.628,Z 700.121,A -85,B 0,C 180,E1 -16772.771,E2 -16772.771} C_VEL
LIN {X 0,Y 296.641,Z 709.988,A -85,B 0,C 180,E1 -16774.652,E2 -16774.652} C_VEL
LIN {X 0,Y 295.016,Z 717.928,A -85,B 0,C 180,E1 -16776.552,E2 -16776.552} C_VEL
LIN {X 0,Y 293.549,Z 724.475,A -85,B 0,C 180,E1 -16778.496,E2 -16778.496} C_VEL
LIN {X 0,Y 292.38,Z 729.78,A -85,B 0,C 180,E1 -16780.466,E2 -16780.466} C_VEL
LIN {X 0,Y 291.403,Z 734.052,A -85,B 0,C 180,E1 -16782.476,E2 -16782.476} C_VEL
LIN {X 0,Y 290.743,Z 737.31,A -85,B 0,C 180,E1 -16784.507,E2 -16784.507} C_VEL
LIN {X 0,Y 289.953,Z 740.208,A -85,B 0,C 180,E1 -16787.261,E2 -16787.261} C_VEL
LIN {X 0,Y 289.651,Z 741.254,A -85,B 0,C 180,E1 -16789.072,E2 -16789.072} C_VEL
LIN {X 0,Y 289.503,Z 741.604,A -85,B 0,C 180,E1 -16790.97,E2 -16790.97} C_VEL
LIN {X 0,Y 289.432,Z 741.045,A -85,B 0,C 180,E1 -16793.254,E2 -16793.254} C_VEL
LIN {X 0,Y 289.636,Z 739.342,A -85,B 0,C 180,E1 -16795.588,E2 -16795.588} C_VEL
LIN {X 0,Y 290.054,Z 736.319,A -85,B 0,C 180,E1 -16797.998,E2 -16797.998} C_VEL
LIN {X 0,Y 290.689,Z 731.747,A -85,B 0,C 180,E1 -16800.501,E2 -16800.501} C_VEL
LIN {X 0,Y 291.485,Z 726.269,A -85,B 0,C 180,E1 -16802.736,E2 -16802.736} C_VEL
LIN {X 0,Y 292.405,Z 720.069,A -85,B 0,C 180,E1 -16804.725,E2 -16804.725} C_VEL
LIN {X 0,Y 293.541,Z 712.263,A -85,B 0,C 180,E1 -16806.732,E2 -16806.732} C_VEL
LIN {X 0,Y 294.761,Z 704.226,A -85,B 0,C 180,E1 -16808.414,E2 -16808.414} C_VEL
LIN {X 0,Y 296.103,Z 694.669,A -85,B 0,C 180,E1 -16810.051,E2 -16810.051} C_VEL
LIN {X 0,Y 297.422,Z 684.191,A -85,B 0,C 180,E1 -16811.503,E2 -16811.503} C_VEL
LIN {X 0,Y 298.626,Z 673.127,A -85,B 0,C 180,E1 -16812.716,E2 -16812.716} C_VEL
LIN {X 0,Y 299.692,Z 660.962,A -85,B 0,C 180,E1 -16813.749,E2 -16813.749} C_VEL
LIN {X 0,Y 300.561,Z 648.143,A -85,B 0,C 180,E1 -16814.547,E2 -16814.547} C_VEL
LIN {X 0,Y 301.139,Z 634.798,A -85,B 0,C 180,E1 -16815.083,E2 -16815.083} C_VEL
LIN {X 0,Y 303.22,Z 563.25,A -85,B 0,C 180,E1 -16816.894,E2 -16816.894} C_VEL
LIN {X 0,Y 296.246,Z 544.461,A -85,B 0,C 180,E1 -16817.955,E2 -16817.955} C_VEL
LIN {X 0,Y 291.633,Z 533.697,A -85,B 0,C 180,E1 -16818.643,E2 -16818.643} C_VEL
LIN {X 0,Y 291.543,Z 533.175,A -85,B 0,C 180,E1 -16818.705,E2 -16818.705} C_VEL
LIN {X 0,Y 291.699,Z 533.15,A -85,B 0,C 180,E1 -16821.688,E2 -16821.688} C_VEL
LIN {X 0,Y 291.626,Z 533.159,A -85,B 0,C 180,E1 -16824.468,E2 -16824.468} C_VEL
LIN {X 0,Y 291.887,Z 533.127,A -85,B 0,C 180,E1 -16828.62,E2 -16828.62} C_VEL
LIN {X 0,Y 291.887,Z 533.126,A -85,B 0,C 180,E1 -16831.38,E2 -16831.38} C_VEL
LIN {X 0,Y 291.744,Z 533.146,A -85,B 0,C 180,E1 -16836.918,E2 -16836.918} C_VEL
LIN {X 0,Y 291.626,Z 533.156,A -85,B 0,C 180,E1 -16839.712,E2 -16839.712} C_VEL
LIN {X 0,Y 291.519,Z 533.168,A -85,B 0,C 180,E1 -16843.95,E2 -16843.95} C_VEL
LIN {X 0,Y 291.484,Z 533.177,A -85,B 0,C 180,E1 -16846.818,E2 -16846.818} C_VEL
LIN {X 0,Y 291.447,Z 533.177,A -85,B 0,C 180,E1 -16849.875,E2 -16849.875} C_VEL
LIN {X 0,Y 291.396,Z 533.184,A -85,B 0,C 180,E1 -16854.205,E2 -16854.205} C_VEL
LIN {X 0,Y 291.419,Z 533.185,A -85,B 0,C 180,E1 -16857.271,E2 -16857.271} C_VEL
LIN {X 0,Y 291.335,Z 533.193,A -85,B 0,C 180,E1 -16860.436,E2 -16860.436} C_VEL
LIN {X 0,Y 291.341,Z 533.192,A -85,B 0,C 180,E1 -16863.698,E2 -16863.698} C_VEL
LIN {X 0,Y 291.4,Z 533.185,A -85,B 0,C 180,E1 -16867.261,E2 -16867.261} C_VEL
LIN {X 0,Y 291.401,Z 533.183,A -85,B 0,C 180,E1 -16870.63,E2 -16870.63} C_VEL
LIN {X 0,Y 291.401,Z 533.184,A -85,B 0,C 180,E1 -16874.379,E2 -16874.379} C_VEL
LIN {X 0,Y 291.382,Z 533.182,A -85,B 0,C 180,E1 -16878.39,E2 -16878.39} C_VEL
LIN {X 0,Y 291.373,Z 533.192,A -85,B 0,C 180,E1 -16881.162,E2 -16881.162} C_VEL
LIN {X 0,Y 291.378,Z 533.188,A -85,B 0,C 180,E1 -16884.629,E2 -16884.629} C_VEL
LIN {X 0,Y 291.316,Z 533.189,A -85,B 0,C 180,E1 -16888.92,E2 -16888.92} C_VEL
LIN {X 0,Y 291.435,Z 533.185,A -85,B 0,C 180,E1 -16893.156,E2 -16893.156} C_VEL
LIN {X 0,Y 291.371,Z 533.184,A -85,B 0,C 180,E1 -16894.924,E2 -16894.924} C_VEL
LIN {X 0,Y 290.681,Z 533.273,A -85,B 0,C 180,E1 -16896.077,E2 -16896.077} C_VEL
LIN {X 0,Y 287.82,Z 533.626,A -85,B 0,C 180,E1 -16897.955,E2 -16897.955} C_VEL
LIN {X 0,Y 285.432,Z 533.925,A -85,B 0,C 180,E1 -16899.48,E2 -16899.48} C_VEL
LIN {X 0,Y 284.443,Z 534.048,A -85,B 0,C 180,E1 -16900.661,E2 -16900.661} C_VEL
LIN {X 0,Y 284.38,Z 534.058,A -85,B 0,C 180,E1 -16901.061,E2 -16901.061} C_VEL
LIN {X 0,Y 284.471,Z 534.047,A -85,B 0,C 180,E1 -16904.47,E2 -16904.47} C_VEL
LIN {X 0,Y 284.483,Z 534.044,A -85,B 0,C 180,E1 -16908.602,E2 -16908.602} C_VEL
LIN {X 0,Y 284.653,Z 534.023,A -85,B 0,C 180,E1 -16911.482,E2 -16911.482} C_VEL
LIN {X 0,Y 284.598,Z 534.03,A -85,B 0,C 180,E1 -16914.332,E2 -16914.332} C_VEL
LIN {X 0,Y 284.85,Z 533.998,A -85,B 0,C 180,E1 -16918.587,E2 -16918.587} C_VEL
LIN {X 0,Y 284.855,Z 534,A -85,B 0,C 180,E1 -16921.414,E2 -16921.414} C_VEL
LIN {X 0,Y 284.596,Z 534.032,A -85,B 0,C 180,E1 -16925.67,E2 -16925.67} C_VEL
LIN {X 0,Y 284.623,Z 534.029,A -85,B 0,C 180,E1 -16929.008,E2 -16929.008} C_VEL
LIN {X 0,Y 284.47,Z 534.049,A -85,B 0,C 180,E1 -16932.848,E2 -16932.848} C_VEL
LIN {X 0,Y 284.483,Z 534.045,A -85,B 0,C 180,E1 -16935.769,E2 -16935.769} C_VEL
LIN {X 0,Y 284.374,Z 534.059,A -85,B 0,C 180,E1 -16940.243,E2 -16940.243} C_VEL
LIN {X 0,Y 284.365,Z 534.059,A -85,B 0,C 180,E1 -16943.876,E2 -16943.876} C_VEL
LIN {X 0,Y 284.394,Z 534.061,A -85,B 0,C 180,E1 -16947.175,E2 -16947.175} C_VEL
LIN {X 0,Y 284.295,Z 534.074,A -85,B 0,C 180,E1 -16951.275,E2 -16951.275} C_VEL
LIN {X 0,Y 284.359,Z 534.066,A -85,B 0,C 180,E1 -16955.355,E2 -16955.355} C_VEL
LIN {X 0,Y 284.314,Z 534.067,A -85,B 0,C 180,E1 -16958.169,E2 -16958.169} C_VEL
LIN {X 0,Y 284.281,Z 534.072,A -85,B 0,C 180,E1 -16962.129,E2 -16962.129} C_VEL
LIN {X 0,Y 284.317,Z 534.067,A -85,B 0,C 180,E1 -16966.203,E2 -16966.203} C_VEL
LIN {X 0,Y 284.351,Z 534.065,A -85,B 0,C 180,E1 -16970.014,E2 -16970.014} C_VEL
LIN {X 0,Y 284.354,Z 534.064,A -85,B 0,C 180,E1 -16974.195,E2 -16974.195} C_VEL
LIN {X 0,Y 284.385,Z 534.179,A -85,B 0,C 180,E1 -16974.486,E2 -16974.486} C_VEL
LIN {X 0,Y 287.196,Z 547.147,A -85,B 0,C 180,E1 -16978.666,E2 -16978.666} C_VEL
LIN {X 0,Y 289.46,Z 558.552,A -85,B 0,C 180,E1 -16982.146,E2 -16982.146} C_VEL
LIN {X 0,Y 289.251,Z 562.171,A -85,B 0,C 180,E1 -16983.083,E2 -16983.083} C_VEL
LIN {X 0,Y 294.623,Z 601.489,A -85,B 0,C 180,E1 -16984.636,E2 -16984.636} C_VEL
LIN {X 0,Y 295.654,Z 610.701,A -85,B 0,C 180,E1 -16984.972,E2 -16984.972} C_VEL
LIN {X 0,Y 293.925,Z 671.256,A -85,B 0,C 180,E1 -16986.577,E2 -16986.577} C_VEL
LIN {X 0,Y 292.99,Z 684.73,A -85,B 0,C 180,E1 -16987.199,E2 -16987.199} C_VEL
LIN {X 0,Y 291.712,Z 697.571,A -85,B 0,C 180,E1 -16988.073,E2 -16988.073} C_VEL
LIN {X 0,Y 290.23,Z 710.146,A -85,B 0,C 180,E1 -16989.259,E2 -16989.259} C_VEL
LIN {X 0,Y 288.671,Z 721.398,A -85,B 0,C 180,E1 -16990.628,E2 -16990.628} C_VEL
LIN {X 0,Y 287.219,Z 731.546,A -85,B 0,C 180,E1 -16992.19,E2 -16992.19} C_VEL
LIN {X 0,Y 285.974,Z 740.071,A -85,B 0,C 180,E1 -16993.805,E2 -16993.805} C_VEL
LIN {X 0,Y 284.757,Z 748.304,A -85,B 0,C 180,E1 -16995.712,E2 -16995.712} C_VEL
LIN {X 0,Y 283.699,Z 755.732,A -85,B 0,C 180,E1 -16997.845,E2 -16997.845} C_VEL
LIN {X 0,Y 283.06,Z 761.678,A -85,B 0,C 180,E1 -16999.991,E2 -16999.991} C_VEL
LIN {X 0,Y 282.671,Z 766.332,A -85,B 0,C 180,E1 -17002.141,E2 -17002.141} C_VEL
LIN {X 0,Y 282.525,Z 769.845,A -85,B 0,C 180,E1 -17004.29,E2 -17004.29} C_VEL
LIN {X 0,Y 282.515,Z 771.583,A -85,B 0,C 180,E1 -17005.72,E2 -17005.72} C_VEL
LIN {X 0,Y 282.519,Z 772.89,A -85,B 0,C 180,E1 -17007.148,E2 -17007.148} C_VEL
LIN {X 0,Y 282.558,Z 773.786,A -85,B 0,C 180,E1 -17008.575,E2 -17008.575} C_VEL
LIN {X 0,Y 282.664,Z 774.262,A -85,B 0,C 180,E1 -17010,E2 -17010} C_VEL
LIN {X 0,Y 282.544,Z 774.277,A -85,B 0,C 180,E1 -17011.425,E2 -17011.425} C_VEL
LIN {X 0,Y 282.493,Z 773.896,A -85,B 0,C 180,E1 -17012.852,E2 -17012.852} C_VEL
LIN {X 0,Y 282.426,Z 772.118,A -85,B 0,C 180,E1 -17015.506,E2 -17015.506} C_VEL
LIN {X 0,Y 282.641,Z 769.323,A -85,B 0,C 180,E1 -17017.86,E2 -17017.86} C_VEL
LIN {X 0,Y 283.071,Z 765.706,A -85,B 0,C 180,E1 -17020.008,E2 -17020.008} C_VEL
LIN {X 0,Y 283.769,Z 760.999,A -85,B 0,C 180,E1 -17022.152,E2 -17022.152} C_VEL
LIN {X 0,Y 285.253,Z 753.936,A -85,B 0,C 180,E1 -17024.627,E2 -17024.627} C_VEL
LIN {X 0,Y 286.821,Z 746.336,A -85,B 0,C 180,E1 -17026.733,E2 -17026.733} C_VEL
LIN {X 0,Y 288.314,Z 738.626,A -85,B 0,C 180,E1 -17028.474,E2 -17028.474} C_VEL
LIN {X 0,Y 290.198,Z 729.332,A -85,B 0,C 180,E1 -17030.188,E2 -17030.188} C_VEL
LIN {X 0,Y 292.22,Z 719.045,A -85,B 0,C 180,E1 -17031.701,E2 -17031.701} C_VEL
LIN {X 0,Y 294.149,Z 707.717,A -85,B 0,C 180,E1 -17033.031,E2 -17033.031} C_VEL
LIN {X 0,Y 295.923,Z 696.055,A -85,B 0,C 180,E1 -17034.091,E2 -17034.091} C_VEL
LIN {X 0,Y 297.493,Z 683.495,A -85,B 0,C 180,E1 -17034.931,E2 -17034.931} C_VEL
LIN {X 0,Y 298.747,Z 669.288,A -85,B 0,C 180,E1 -17035.572,E2 -17035.572} C_VEL
LIN {X 0,Y 300.869,Z 610.843,A -85,B 0,C 180,E1 -17037.148,E2 -17037.148} C_VEL
LIN {X 0,Y 298.2,Z 589.177,A -85,B 0,C 180,E1 -17038.146,E2 -17038.146} C_VEL
LIN {X 0,Y 294.325,Z 568.281,A -85,B 0,C 180,E1 -17039.308,E2 -17039.308} C_VEL
LIN {X 0,Y 290.27,Z 558.905,A -85,B 0,C 180,E1 -17040.192,E2 -17040.192} C_VEL
LIN {X 0,Y 288.041,Z 548.25,A -85,B 0,C 180,E1 -17043.944,E2 -17043.944} C_VEL
LIN {X 0,Y 285.654,Z 538.768,A -85,B 0,C 180,E1 -17047.635,E2 -17047.635} C_VEL
LIN {X 0,Y 284.38,Z 534.062,A -85,B 0,C 180,E1 -17049.671,E2 -17049.671} C_VEL
LIN {X 0,Y 284.318,Z 534.07,A -85,B 0,C 180,E1 -17053.797,E2 -17053.797} C_VEL
LIN {X 0,Y 284.28,Z 534.07,A -85,B 0,C 180,E1 -17058.125,E2 -17058.125} C_VEL
LIN {X 0,Y 284.333,Z 534.066,A -85,B 0,C 180,E1 -17062.274,E2 -17062.274} C_VEL
LIN {X 0,Y 284.321,Z 534.064,A -85,B 0,C 180,E1 -17065.352,E2 -17065.352} C_VEL
LIN {X 0,Y 284.292,Z 534.068,A -85,B 0,C 180,E1 -17068.725,E2 -17068.725} C_VEL
LIN {X 0,Y 284.394,Z 534.054,A -85,B 0,C 180,E1 -17072.825,E2 -17072.825} C_VEL
LIN {X 0,Y 284.362,Z 534.059,A -85,B 0,C 180,E1 -17076.706,E2 -17076.706} C_VEL
LIN {X 0,Y 284.399,Z 534.059,A -85,B 0,C 180,E1 -17081.261,E2 -17081.261} C_VEL
LIN {X 0,Y 284.487,Z 534.048,A -85,B 0,C 180,E1 -17084.458,E2 -17084.458} C_VEL
LIN {X 0,Y 284.482,Z 534.05,A -85,B 0,C 180,E1 -17088.601,E2 -17088.601} C_VEL
LIN {X 0,Y 284.652,Z 534.028,A -85,B 0,C 180,E1 -17091.48,E2 -17091.48} C_VEL
LIN {X 0,Y 284.596,Z 534.028,A -85,B 0,C 180,E1 -17094.33,E2 -17094.33} C_VEL
LIN {X 0,Y 284.85,Z 534.002,A -85,B 0,C 180,E1 -17098.586,E2 -17098.586} C_VEL
LIN {X 0,Y 284.853,Z 534.001,A -85,B 0,C 180,E1 -17101.413,E2 -17101.413} C_VEL
LIN {X 0,Y 284.681,Z 534.022,A -85,B 0,C 180,E1 -17107.09,E2 -17107.09} C_VEL
LIN {X 0,Y 284.512,Z 534.046,A -85,B 0,C 180,E1 -17109.957,E2 -17109.957} C_VEL
LIN {X 0,Y 284.471,Z 534.051,A -85,B 0,C 180,E1 -17114.303,E2 -17114.303} C_VEL
LIN {X 0,Y 284.418,Z 534.057,A -85,B 0,C 180,E1 -17117.248,E2 -17117.248} C_VEL
LIN {X 0,Y 284.343,Z 534.133,A -85,B 0,C 180,E1 -17120.716,E2 -17120.716} C_VEL
LIN {X 0,Y 284.461,Z 534.817,A -85,B 0,C 180,E1 -17121.039,E2 -17121.039} C_VEL
LIN {X 0,Y 285.825,Z 537.625,A -85,B 0,C 180,E1 -17121.359,E2 -17121.359} C_VEL
LIN {X 0,Y 291.02,Z 546.325,A -85,B 0,C 180,E1 -17122.42,E2 -17122.42} C_VEL
LIN {X 0,Y 297.625,Z 559.526,A -85,B 0,C 180,E1 -17123.754,E2 -17123.754} C_VEL
LIN {X 0,Y 302.161,Z 570.179,A -85,B 0,C 180,E1 -17124.658,E2 -17124.658} C_VEL
LIN {X 0,Y 299.484,Z 640.973,A -85,B 0,C 180,E1 -17126.57,E2 -17126.57} C_VEL
LIN {X 0,Y 298.51,Z 654.491,A -85,B 0,C 180,E1 -17127.215,E2 -17127.215} C_VEL
LIN {X 0,Y 297.297,Z 667.263,A -85,B 0,C 180,E1 -17128.127,E2 -17128.127} C_VEL
LIN {X 0,Y 295.731,Z 679.446,A -85,B 0,C 180,E1 -17129.297,E2 -17129.297} C_VEL
LIN {X 0,Y 294.027,Z 690.298,A -85,B 0,C 180,E1 -17130.631,E2 -17130.631} C_VEL
LIN {X 0,Y 292.118,Z 700.571,A -85,B 0,C 180,E1 -17132.223,E2 -17132.223} C_VEL
LIN {X 0,Y 290.051,Z 710.363,A -85,B 0,C 180,E1 -17134.127,E2 -17134.127} C_VEL
LIN {X 0,Y 288.324,Z 718.356,A -85,B 0,C 180,E1 -17136.077,E2 -17136.077} C_VEL
LIN {X 0,Y 286.609,Z 725.592,A -85,B 0,C 180,E1 -17138.311,E2 -17138.311} C_VEL
LIN {X 0,Y 285.415,Z 730.564,A -85,B 0,C 180,E1 -17140.242,E2 -17140.242} C_VEL
LIN {X 0,Y 284.455,Z 734.516,A -85,B 0,C 180,E1 -17142.167,E2 -17142.167} C_VEL
LIN {X 0,Y 283.796,Z 737.551,A -85,B 0,C 180,E1 -17144.098,E2 -17144.098} C_VEL
LIN {X 0,Y 283.178,Z 739.769,A -85,B 0,C 180,E1 -17146.031,E2 -17146.031} C_VEL
LIN {X 0,Y 282.689,Z 741.364,A -85,B 0,C 180,E1 -17148.23,E2 -17148.23} C_VEL
LIN {X 0,Y 282.431,Z 741.997,A -85,B 0,C 180,E1 -17150.479,E2 -17150.479} C_VEL
LIN {X 0,Y 282.367,Z 741.397,A -85,B 0,C 180,E1 -17153.321,E2 -17153.321} C_VEL
LIN {X 0,Y 282.5,Z 740.1,A -85,B 0,C 180,E1 -17155.181,E2 -17155.181} C_VEL
LIN {X 0,Y 282.875,Z 737.333,A -85,B 0,C 180,E1 -17157.641,E2 -17157.641} C_VEL
LIN {X 0,Y 283.525,Z 732.836,A -85,B 0,C 180,E1 -17160.281,E2 -17160.281} C_VEL
LIN {X 0,Y 284.412,Z 726.891,A -85,B 0,C 180,E1 -17162.819,E2 -17162.819} C_VEL
LIN {X 0,Y 285.372,Z 720.733,A -85,B 0,C 180,E1 -17164.861,E2 -17164.861} C_VEL
LIN {X 0,Y 286.533,Z 713.089,A -85,B 0,C 180,E1 -17166.894,E2 -17166.894} C_VEL
LIN {X 0,Y 287.978,Z 703.657,A -85,B 0,C 180,E1 -17168.902,E2 -17168.902} C_VEL
LIN {X 0,Y 289.402,Z 693.564,A -85,B 0,C 180,E1 -17170.629,E2 -17170.629} C_VEL
LIN {X 0,Y 290.789,Z 683.095,A -85,B 0,C 180,E1 -17172.053,E2 -17172.053} C_VEL
LIN {X 0,Y 292.164,Z 670.441,A -85,B 0,C 180,E1 -17173.41,E2 -17173.41} C_VEL
LIN {X 0,Y 293.234,Z 658.308,A -85,B 0,C 180,E1 -17174.387,E2 -17174.387} C_VEL
LIN {X 0,Y 294.016,Z 645.432,A -85,B 0,C 180,E1 -17175.133,E2 -17175.133} C_VEL
LIN {X 0,Y 294.571,Z 632.019,A -85,B 0,C 180,E1 -17175.625,E2 -17175.625} C_VEL
LIN {X 0,Y 296.585,Z 564.763,A -85,B 0,C 180,E1 -17177.354,E2 -17177.354} C_VEL
LIN {X 0,Y 290.022,Z 547.13,A -85,B 0,C 180,E1 -17178.388,E2 -17178.388} C_VEL
LIN {X 0,Y 284.669,Z 534.872,A -85,B 0,C 180,E1 -17179.209,E2 -17179.209} C_VEL
LIN {X 0,Y 284.506,Z 534.05,A -85,B 0,C 180,E1 -17179.284,E2 -17179.284} C_VEL
LIN {X 0,Y 284.69,Z 534.025,A -85,B 0,C 180,E1 -17182.91,E2 -17182.91} C_VEL
LIN {X 0,Y 284.853,Z 534.003,A -85,B 0,C 180,E1 -17188.586,E2 -17188.586} C_VEL
LIN {X 0,Y 284.853,Z 534.002,A -85,B 0,C 180,E1 -17191.414,E2 -17191.414} C_VEL
LIN {X 0,Y 284.696,Z 534.023,A -85,B 0,C 180,E1 -17197.09,E2 -17197.09} C_VEL
LIN {X 0,Y 284.563,Z 534.036,A -85,B 0,C 180,E1 -17199.955,E2 -17199.955} C_VEL
LIN {X 0,Y 284.478,Z 534.046,A -85,B 0,C 180,E1 -17204.303,E2 -17204.303} C_VEL
LIN {X 0,Y 284.422,Z 534.055,A -85,B 0,C 180,E1 -17207.248,E2 -17207.248} C_VEL
LIN {X 0,Y 284.375,Z 534.058,A -85,B 0,C 180,E1 -17210.242,E2 -17210.242} C_VEL
LIN {X 0,Y 284.365,Z 534.06,A -85,B 0,C 180,E1 -17213.875,E2 -17213.875} C_VEL
LIN {X 0,Y 284.393,Z 534.061,A -85,B 0,C 180,E1 -17217.173,E2 -17217.173} C_VEL
LIN {X 0,Y 284.294,Z 534.072,A -85,B 0,C 180,E1 -17221.274,E2 -17221.274} C_VEL
LIN {X 0,Y 284.357,Z 534.064,A -85,B 0,C 180,E1 -17225.354,E2 -17225.354} C_VEL
LIN {X 0,Y 284.332,Z 534.062,A -85,B 0,C 180,E1 -17228.165,E2 -17228.165} C_VEL
LIN {X 0,Y 284.339,Z 534.063,A -85,B 0,C 180,E1 -17232.141,E2 -17232.141} C_VEL
LIN {X 0,Y 284.347,Z 534.061,A -85,B 0,C 180,E1 -17236.208,E2 -17236.208} C_VEL
LIN {X 0,Y 284.345,Z 534.061,A -85,B 0,C 180,E1 -17240.013,E2 -17240.013} C_VEL
LIN {X 0,Y 284.345,Z 534.063,A -85,B 0,C 180,E1 -17243.617,E2 -17243.617} C_VEL
LIN {X 0,Y 284.301,Z 534.067,A -85,B 0,C 180,E1 -17247.19,E2 -17247.19} C_VEL
LIN {X 0,Y 284.352,Z 534.06,A -85,B 0,C 180,E1 -17250.376,E2 -17250.376} C_VEL
LIN {X 0,Y 284.373,Z 534.061,A -85,B 0,C 180,E1 -17253.587,E2 -17253.587} C_VEL
LIN {X 0,Y 284.326,Z 534.066,A -85,B 0,C 180,E1 -17256.704,E2 -17256.704} C_VEL
LIN {X 0,Y 284.38,Z 534.058,A -85,B 0,C 180,E1 -17261.061,E2 -17261.061} C_VEL
LIN {X 0,Y 283.764,Z 534.144,A -85,B 0,C 180,E1 -17262.244,E2 -17262.244} C_VEL
LIN {X 0,Y 280.942,Z 534.499,A -85,B 0,C 180,E1 -17264.171,E2 -17264.171} C_VEL
LIN {X 0,Y 278.519,Z 534.794,A -85,B 0,C 180,E1 -17265.737,E2 -17265.737} C_VEL
LIN {X 0,Y 277.479,Z 534.921,A -85,B 0,C 180,E1 -17266.95,E2 -17266.95} C_VEL
LIN {X 0,Y 277.395,Z 534.926,A -85,B 0,C 180,E1 -17267.362,E2 -17267.362} C_VEL
LIN {X 0,Y 277.609,Z 534.9,A -85,B 0,C 180,E1 -17271.264,E2 -17271.264} C_VEL
LIN {X 0,Y 277.568,Z 534.905,A -85,B 0,C 180,E1 -17274.188,E2 -17274.188} C_VEL
LIN {X 0,Y 277.816,Z 534.874,A -85,B 0,C 180,E1 -17278.551,E2 -17278.551} C_VEL
LIN {X 0,Y 277.821,Z 534.875,A -85,B 0,C 180,E1 -17281.45,E2 -17281.45} C_VEL
LIN {X 0,Y 277.566,Z 534.907,A -85,B 0,C 180,E1 -17285.814,E2 -17285.814} C_VEL
LIN {X 0,Y 277.564,Z 534.908,A -85,B 0,C 180,E1 -17289.081,E2 -17289.081} C_VEL
LIN {X 0,Y 277.411,Z 534.93,A -85,B 0,C 180,E1 -17293.181,E2 -17293.181} C_VEL
LIN {X 0,Y 277.401,Z 534.926,A -85,B 0,C 180,E1 -17296.183,E2 -17296.183} C_VEL
LIN {X 0,Y 277.341,Z 534.936,A -85,B 0,C 180,E1 -17300.351,E2 -17300.351} C_VEL
LIN {X 0,Y 277.315,Z 534.936,A -85,B 0,C 180,E1 -17304.171,E2 -17304.171} C_VEL
LIN {X 0,Y 277.322,Z 534.941,A -85,B 0,C 180,E1 -17307.506,E2 -17307.506} C_VEL
LIN {X 0,Y 277.269,Z 534.944,A -85,B 0,C 180,E1 -17310.483,E2 -17310.483} C_VEL
LIN {X 0,Y 277.252,Z 534.947,A -85,B 0,C 180,E1 -17313.896,E2 -17313.896} C_VEL
LIN {X 0,Y 277.275,Z 534.947,A -85,B 0,C 180,E1 -17317.469,E2 -17317.469} C_VEL
LIN {X 0,Y 277.214,Z 534.955,A -85,B 0,C 180,E1 -17321.237,E2 -17321.237} C_VEL
LIN {X 0,Y 277.246,Z 534.951,A -85,B 0,C 180,E1 -17325.218,E2 -17325.218} C_VEL
LIN {X 0,Y 277.295,Z 534.946,A -85,B 0,C 180,E1 -17329.496,E2 -17329.496} C_VEL
LIN {X 0,Y 277.314,Z 534.978,A -85,B 0,C 180,E1 -17333.987,E2 -17333.987} C_VEL
LIN {X 0,Y 279.751,Z 546.232,A -85,B 0,C 180,E1 -17337.735,E2 -17337.735} C_VEL
LIN {X 0,Y 282.096,Z 557.466,A -85,B 0,C 180,E1 -17341.292,E2 -17341.292} C_VEL
LIN {X 0,Y 282.451,Z 561.487,A -85,B 0,C 180,E1 -17342.492,E2 -17342.492} C_VEL
LIN {X 0,Y 287.765,Z 600.569,A -85,B 0,C 180,E1 -17344.086,E2 -17344.086} C_VEL
LIN {X 0,Y 289.021,Z 611.053,A -85,B 0,C 180,E1 -17344.487,E2 -17344.487} C_VEL
LIN {X 0,Y 287.252,Z 670.47,A -85,B 0,C 180,E1 -17346.095,E2 -17346.095} C_VEL
LIN {X 0,Y 286.284,Z 684.055,A -85,B 0,C 180,E1 -17346.729,E2 -17346.729} C_VEL
LIN {X 0,Y 284.979,Z 696.985,A -85,B 0,C 180,E1 -17347.623,E2 -17347.623} C_VEL
LIN {X 0,Y 283.545,Z 708.805,A -85,B 0,C 180,E1 -17348.747,E2 -17348.747} C_VEL
LIN {X 0,Y 281.998,Z 720.239,A -85,B 0,C 180,E1 -17350.15,E2 -17350.15} C_VEL
LIN {X 0,Y 280.546,Z 729.491,A -85,B 0,C 180,E1 -17351.563,E2 -17351.563} C_VEL
LIN {X 0,Y 279.075,Z 738.73,A -85,B 0,C 180,E1 -17353.294,E2 -17353.294} C_VEL
LIN {X 0,Y 278.033,Z 746.108,A -85,B 0,C 180,E1 -17354.984,E2 -17354.984} C_VEL
LIN {X 0,Y 276.89,Z 753.864,A -85,B 0,C 180,E1 -17357.168,E2 -17357.168} C_VEL
LIN {X 0,Y 276.2,Z 759.161,A -85,B 0,C 180,E1 -17358.998,E2 -17358.998} C_VEL
LIN {X 0,Y 275.7,Z 764.274,A -85,B 0,C 180,E1 -17361.202,E2 -17361.202} C_VEL
LIN {X 0,Y 275.455,Z 768.208,A -85,B 0,C 180,E1 -17363.407,E2 -17363.407} C_VEL
LIN {X 0,Y 275.435,Z 771.071,A -85,B 0,C 180,E1 -17365.61,E2 -17365.61} C_VEL
LIN {X 0,Y 275.444,Z 772.402,A -85,B 0,C 180,E1 -17367.075,E2 -17367.075} C_VEL
LIN {X 0,Y 275.472,Z 773.319,A -85,B 0,C 180,E1 -17368.538,E2 -17368.538} C_VEL
LIN {X 0,Y 275.575,Z 773.83,A -85,B 0,C 180,E1 -17370,E2 -17370} C_VEL
LIN {X 0,Y 275.458,Z 773.875,A -85,B 0,C 180,E1 -17371.462,E2 -17371.462} C_VEL
LIN {X 0,Y 275.416,Z 773.514,A -85,B 0,C 180,E1 -17372.925,E2 -17372.925} C_VEL
LIN {X 0,Y 275.352,Z 771.918,A -85,B 0,C 180,E1 -17375.477,E2 -17375.477} C_VEL
LIN {X 0,Y 275.567,Z 769.025,A -85,B 0,C 180,E1 -17378.063,E2 -17378.063} C_VEL
LIN {X 0,Y 276.026,Z 765.459,A -85,B 0,C 180,E1 -17380.266,E2 -17380.266} C_VEL
LIN {X 0,Y 276.808,Z 760.816,A -85,B 0,C 180,E1 -17382.463,E2 -17382.463} C_VEL
LIN {X 0,Y 278.37,Z 753.845,A -85,B 0,C 180,E1 -17384.997,E2 -17384.997} C_VEL
LIN {X 0,Y 280.012,Z 746.309,A -85,B 0,C 180,E1 -17387.152,E2 -17387.152} C_VEL
LIN {X 0,Y 281.935,Z 737.003,A -85,B 0,C 180,E1 -17389.286,E2 -17389.286} C_VEL
LIN {X 0,Y 284.198,Z 726.303,A -85,B 0,C 180,E1 -17391.202,E2 -17391.202} C_VEL
LIN {X 0,Y 286.375,Z 715.492,A -85,B 0,C 180,E1 -17392.738,E2 -17392.738} C_VEL
LIN {X 0,Y 288.229,Z 705.073,A -85,B 0,C 180,E1 -17393.914,E2 -17393.914} C_VEL
LIN {X 0,Y 290.082,Z 692.684,A -85,B 0,C 180,E1 -17394.99,E2 -17394.99} C_VEL
LIN {X 0,Y 291.77,Z 679.14,A -85,B 0,C 180,E1 -17395.835,E2 -17395.835} C_VEL
LIN {X 0,Y 292.806,Z 666.686,A -85,B 0,C 180,E1 -17396.346,E2 -17396.346} C_VEL
LIN {X 0,Y 294.796,Z 611.363,A -85,B 0,C 180,E1 -17397.863,E2 -17397.863} C_VEL
LIN {X 0,Y 291.889,Z 588.095,A -85,B 0,C 180,E1 -17398.982,E2 -17398.982} C_VEL
LIN {X 0,Y 288.618,Z 570.839,A -85,B 0,C 180,E1 -17400.006,E2 -17400.006} C_VEL
LIN {X 0,Y 284.234,Z 561.368,A -85,B 0,C 180,E1 -17400.967,E2 -17400.967} C_VEL
LIN {X 0,Y 283.018,Z 558.245,A -85,B 0,C 180,E1 -17401.308,E2 -17401.308} C_VEL
LIN {X 0,Y 281.209,Z 549.752,A -85,B 0,C 180,E1 -17404.437,E2 -17404.437} C_VEL
LIN {X 0,Y 278.976,Z 540.847,A -85,B 0,C 180,E1 -17408.032,E2 -17408.032} C_VEL
LIN {X 0,Y 277.269,Z 534.945,A -85,B 0,C 180,E1 -17410.697,E2 -17410.697} C_VEL
LIN {X 0,Y 277.246,Z 534.948,A -85,B 0,C 180,E1 -17414.782,E2 -17414.782} C_VEL
LIN {X 0,Y 277.214,Z 534.954,A -85,B 0,C 180,E1 -17418.763,E2 -17418.763} C_VEL
LIN {X 0,Y 277.279,Z 534.942,A -85,B 0,C 180,E1 -17422.532,E2 -17422.532} C_VEL
LIN {X 0,Y 277.251,Z 534.943,A -85,B 0,C 180,E1 -17426.104,E2 -17426.104} C_VEL
LIN {X 0,Y 277.259,Z 534.944,A -85,B 0,C 180,E1 -17429.537,E2 -17429.537} C_VEL
LIN {X 0,Y 277.355,Z 534.931,A -85,B 0,C 180,E1 -17432.863,E2 -17432.863} C_VEL
LIN {X 0,Y 277.324,Z 534.932,A -85,B 0,C 180,E1 -17436.078,E2 -17436.078} C_VEL
LIN {X 0,Y 277.34,Z 534.938,A -85,B 0,C 180,E1 -17440.765,E2 -17440.765} C_VEL
LIN {X 0,Y 277.429,Z 534.925,A -85,B 0,C 180,E1 -17445.325,E2 -17445.325} C_VEL
LIN {X 0,Y 277.501,Z 534.911,A -85,B 0,C 180,E1 -17449.788,E2 -17449.788} C_VEL
LIN {X 0,Y 277.645,Z 534.898,A -85,B 0,C 180,E1 -17452.728,E2 -17452.728} C_VEL
LIN {X 0,Y 277.816,Z 534.878,A -85,B 0,C 180,E1 -17458.55,E2 -17458.55} C_VEL
LIN {X 0,Y 277.819,Z 534.878,A -85,B 0,C 180,E1 -17461.449,E2 -17461.449} C_VEL
LIN {X 0,Y 277.635,Z 534.901,A -85,B 0,C 180,E1 -17467.271,E2 -17467.271} C_VEL
LIN {X 0,Y 277.454,Z 534.925,A -85,B 0,C 180,E1 -17470.212,E2 -17470.212} C_VEL
LIN {X 0,Y 277.421,Z 534.931,A -85,B 0,C 180,E1 -17474.674,E2 -17474.674} C_VEL
LIN {X 0,Y 277.336,Z 534.938,A -85,B 0,C 180,E1 -17479.234,E2 -17479.234} C_VEL
LIN {X 0,Y 277.373,Z 535.176,A -85,B 0,C 180,E1 -17479.812,E2 -17479.812} C_VEL
LIN {X 0,Y 277.478,Z 535.759,A -85,B 0,C 180,E1 -17479.95,E2 -17479.95} C_VEL
LIN {X 0,Y 278.843,Z 538.522,A -85,B 0,C 180,E1 -17480.28,E2 -17480.28} C_VEL
LIN {X 0,Y 280.021,Z 540.14,A -85,B 0,C 180,E1 -17480.533,E2 -17480.533} C_VEL
LIN {X 0,Y 286.676,Z 551.682,A -85,B 0,C 180,E1 -17481.975,E2 -17481.975} C_VEL
LIN {X 0,Y 293.021,Z 564.69,A -85,B 0,C 180,E1 -17483.312,E2 -17483.312} C_VEL
LIN {X 0,Y 296.252,Z 572.328,A -85,B 0,C 180,E1 -17483.987,E2 -17483.987} C_VEL
LIN {X 0,Y 293.397,Z 641.376,A -85,B 0,C 180,E1 -17485.874,E2 -17485.874} C_VEL
LIN {X 0,Y 292.364,Z 655.191,A -85,B 0,C 180,E1 -17486.548,E2 -17486.548} C_VEL
LIN {X 0,Y 291.224,Z 666.851,A -85,B 0,C 180,E1 -17487.388,E2 -17487.388} C_VEL
LIN {X 0,Y 289.593,Z 678.968,A -85,B 0,C 180,E1 -17488.552,E2 -17488.552} C_VEL
LIN {X 0,Y 287.908,Z 689.328,A -85,B 0,C 180,E1 -17489.825,E2 -17489.825} C_VEL
LIN {X 0,Y 285.902,Z 699.781,A -85,B 0,C 180,E1 -17491.425,E2 -17491.425} C_VEL
LIN {X 0,Y 284.181,Z 707.884,A -85,B 0,C 180,E1 -17492.961,E2 -17492.961} C_VEL
LIN {X 0,Y 282.192,Z 716.418,A -85,B 0,C 180,E1 -17494.946,E2 -17494.946} C_VEL
LIN {X 0,Y 280.5,Z 723.374,A -85,B 0,C 180,E1 -17496.964,E2 -17496.964} C_VEL
LIN {X 0,Y 279.031,Z 729.08,A -85,B 0,C 180,E1 -17499.025,E2 -17499.025} C_VEL
LIN {X 0,Y 277.884,Z 733.64,A -85,B 0,C 180,E1 -17501.114,E2 -17501.114} C_VEL
LIN {X 0,Y 276.984,Z 737.21,A -85,B 0,C 180,E1 -17503.241,E2 -17503.241} C_VEL
LIN {X 0,Y 276.256,Z 739.863,A -85,B 0,C 180,E1 -17505.423,E2 -17505.423} C_VEL
LIN {X 0,Y 275.716,Z 741.6,A -85,B 0,C 180,E1 -17507.663,E2 -17507.663} C_VEL
LIN {X 0,Y 275.353,Z 742.416,A -85,B 0,C 180,E1 -17510.352,E2 -17510.352} C_VEL
LIN {X 0,Y 275.269,Z 742.17,A -85,B 0,C 180,E1 -17512.322,E2 -17512.322} C_VEL
LIN {X 0,Y 275.356,Z 740.841,A -85,B 0,C 180,E1 -17514.759,E2 -17514.759} C_VEL
LIN {X 0,Y 275.802,Z 737.788,A -85,B 0,C 180,E1 -17517.649,E2 -17517.649} C_VEL
LIN {X 0,Y 276.342,Z 734.289,A -85,B 0,C 180,E1 -17519.847,E2 -17519.847} C_VEL
LIN {X 0,Y 276.977,Z 729.984,A -85,B 0,C 180,E1 -17521.909,E2 -17521.909} C_VEL
LIN {X 0,Y 277.899,Z 724.102,A -85,B 0,C 180,E1 -17524.136,E2 -17524.136} C_VEL
LIN {X 0,Y 279.013,Z 717.118,A -85,B 0,C 180,E1 -17526.233,E2 -17526.233} C_VEL
LIN {X 0,Y 280.497,Z 708.018,A -85,B 0,C 180,E1 -17528.412,E2 -17528.412} C_VEL
LIN {X 0,Y 281.987,Z 698.106,A -85,B 0,C 180,E1 -17530.31,E2 -17530.31} C_VEL
LIN {X 0,Y 283.492,Z 687.3,A -85,B 0,C 180,E1 -17531.948,E2 -17531.948} C_VEL
LIN {X 0,Y 284.918,Z 675.59,A -85,B 0,C 180,E1 -17533.356,E2 -17533.356} C_VEL
LIN {X 0,Y 286.123,Z 663.031,A -85,B 0,C 180,E1 -17534.507,E2 -17534.507} C_VEL
LIN {X 0,Y 287.027,Z 650.155,A -85,B 0,C 180,E1 -17535.374,E2 -17535.374} C_VEL
LIN {X 0,Y 287.717,Z 637.193,A -85,B 0,C 180,E1 -17535.952,E2 -17535.952} C_VEL
LIN {X 0,Y 289.947,Z 566.18,A -85,B 0,C 180,E1 -17537.841,E2 -17537.841} C_VEL
LIN {X 0,Y 283.998,Z 550.229,A -85,B 0,C 180,E1 -17538.807,E2 -17538.807} C_VEL
LIN {X 0,Y 277.6,Z 535.431,A -85,B 0,C 180,E1 -17539.815,E2 -17539.815} C_VEL
LIN {X 0,Y 277.513,Z 534.92,A -85,B 0,C 180,E1 -17539.881,E2 -17539.881} C_VEL
LIN {X 0,Y 277.645,Z 534.902,A -85,B 0,C 180,E1 -17542.729,E2 -17542.729} C_VEL
LIN {X 0,Y 277.819,Z 534.879,A -85,B 0,C 180,E1 -17548.55,E2 -17548.55} C_VEL
LIN {X 0,Y 277.819,Z 534.878,A -85,B 0,C 180,E1 -17551.45,E2 -17551.45} C_VEL
LIN {X 0,Y 277.65,Z 534.9,A -85,B 0,C 180,E1 -17557.271,E2 -17557.271} C_VEL
LIN {X 0,Y 277.504,Z 534.915,A -85,B 0,C 180,E1 -17560.211,E2 -17560.211} C_VEL
LIN {X 0,Y 277.431,Z 534.926,A -85,B 0,C 180,E1 -17564.674,E2 -17564.674} C_VEL
LIN {X 0,Y 277.342,Z 534.937,A -85,B 0,C 180,E1 -17569.234,E2 -17569.234} C_VEL
LIN {X 0,Y 277.315,Z 534.938,A -85,B 0,C 180,E1 -17574.17,E2 -17574.17} C_VEL
LIN {X 0,Y 277.322,Z 534.939,A -85,B 0,C 180,E1 -17577.505,E2 -17577.505} C_VEL
LIN {X 0,Y 277.267,Z 534.945,A -85,B 0,C 180,E1 -17580.481,E2 -17580.481} C_VEL
LIN {X 0,Y 277.25,Z 534.947,A -85,B 0,C 180,E1 -17583.894,E2 -17583.894} C_VEL
LIN {X 0,Y 277.286,Z 534.941,A -85,B 0,C 180,E1 -17587.465,E2 -17587.465} C_VEL
LIN {X 0,Y 277.289,Z 534.945,A -85,B 0,C 180,E1 -17591.221,E2 -17591.221} C_VEL
LIN {X 0,Y 277.282,Z 534.944,A -85,B 0,C 180,E1 -17595.208,E2 -17595.208} C_VEL
LIN {X 0,Y 277.289,Z 534.941,A -85,B 0,C 180,E1 -17599.494,E2 -17599.494} C_VEL
LIN {X 0,Y 277.28,Z 534.944,A -85,B 0,C 180,E1 -17602.534,E2 -17602.534} C_VEL
LIN {X 0,Y 277.247,Z 534.944,A -85,B 0,C 180,E1 -17606.105,E2 -17606.105} C_VEL
LIN {X 0,Y 277.255,Z 534.945,A -85,B 0,C 180,E1 -17609.539,E2 -17609.539} C_VEL
LIN {X 0,Y 277.354,Z 534.936,A -85,B 0,C 180,E1 -17612.865,E2 -17612.865} C_VEL
LIN {X 0,Y 277.29,Z 534.94,A -85,B 0,C 180,E1 -17616.077,E2 -17616.077} C_VEL
LIN {X 0,Y 277.336,Z 534.932,A -85,B 0,C 180,E1 -17620.766,E2 -17620.766} C_VEL
LIN {X 0,Y 277.422,Z 534.928,A -85,B 0,C 180,E1 -17625.326,E2 -17625.326} C_VEL
LIN {X 0,Y 277.395,Z 534.926,A -85,B 0,C 180,E1 -17627.362,E2 -17627.362} C_VEL
LIN {X 0,Y 276.749,Z 535.008,A -85,B 0,C 180,E1 -17628.575,E2 -17628.575} C_VEL
LIN {X 0,Y 273.973,Z 535.347,A -85,B 0,C 180,E1 -17630.555,E2 -17630.555} C_VEL
LIN {X 0,Y 271.62,Z 535.644,A -85,B 0,C 180,E1 -17632.163,E2 -17632.163} C_VEL
LIN {X 0,Y 270.616,Z 535.774,A -85,B 0,C 180,E1 -17633.407,E2 -17633.407} C_VEL
LIN {X 0,Y 270.537,Z 535.779,A -85,B 0,C 180,E1 -17633.828,E2 -17633.828} C_VEL
LIN {X 0,Y 270.782,Z 535.75,A -85,B 0,C 180,E1 -17638.513,E2 -17638.513} C_VEL
LIN {X 0,Y 270.787,Z 535.751,A -85,B 0,C 180,E1 -17641.488,E2 -17641.488} C_VEL
LIN {X 0,Y 270.536,Z 535.782,A -85,B 0,C 180,E1 -17645.965,E2 -17645.965} C_VEL
LIN {X 0,Y 270.519,Z 535.784,A -85,B 0,C 180,E1 -17649.176,E2 -17649.176} C_VEL
LIN {X 0,Y 270.354,Z 535.808,A -85,B 0,C 180,E1 -17653.531,E2 -17653.531} C_VEL
LIN {X 0,Y 270.35,Z 535.805,A -85,B 0,C 180,E1 -17656.617,E2 -17656.617} C_VEL
LIN {X 0,Y 270.288,Z 535.815,A -85,B 0,C 180,E1 -17660.602,E2 -17660.602} C_VEL
LIN {X 0,Y 270.27,Z 535.814,A -85,B 0,C 180,E1 -17664.587,E2 -17664.587} C_VEL
LIN {X 0,Y 270.269,Z 535.817,A -85,B 0,C 180,E1 -17667.91,E2 -17667.91} C_VEL
LIN {X 0,Y 270.182,Z 535.832,A -85,B 0,C 180,E1 -17671.349,E2 -17671.349} C_VEL
LIN {X 0,Y 270.212,Z 535.824,A -85,B 0,C 180,E1 -17674.905,E2 -17674.905} C_VEL
LIN {X 0,Y 270.196,Z 535.827,A -85,B 0,C 180,E1 -17678.712,E2 -17678.712} C_VEL
LIN {X 0,Y 270.188,Z 535.83,A -85,B 0,C 180,E1 -17683.255,E2 -17683.255} C_VEL
LIN {X 0,Y 270.222,Z 535.828,A -85,B 0,C 180,E1 -17687.453,E2 -17687.453} C_VEL
LIN {X 0,Y 270.245,Z 535.822,A -85,B 0,C 180,E1 -17691.382,E2 -17691.382} C_VEL
LIN {X 0,Y 270.315,Z 535.919,A -85,B 0,C 180,E1 -17693.528,E2 -17693.528} C_VEL
LIN {X 0,Y 273.033,Z 548.583,A -85,B 0,C 180,E1 -17697.846,E2 -17697.846} C_VEL
LIN {X 0,Y 275.338,Z 559.909,A -85,B 0,C 180,E1 -17701.505,E2 -17701.505} C_VEL
LIN {X 0,Y 275.57,Z 561.37,A -85,B 0,C 180,E1 -17701.89,E2 -17701.89} C_VEL
LIN {X 0,Y 278.602,Z 581.461,A -85,B 0,C 180,E1 -17702.768,E2 -17702.768} C_VEL
LIN {X 0,Y 282.41,Z 611.46,A -85,B 0,C 180,E1 -17703.981,E2 -17703.981} C_VEL
LIN {X 0,Y 280.547,Z 670.782,A -85,B 0,C 180,E1 -17705.635,E2 -17705.635} C_VEL
LIN {X 0,Y 279.539,Z 684.128,A -85,B 0,C 180,E1 -17706.281,E2 -17706.281} C_VEL
LIN {X 0,Y 278.265,Z 696.393,A -85,B 0,C 180,E1 -17707.151,E2 -17707.151} C_VEL
LIN {X 0,Y 276.894,Z 707.466,A -85,B 0,C 180,E1 -17708.211,E2 -17708.211} C_VEL
LIN {X 0,Y 275.25,Z 719.063,A -85,B 0,C 180,E1 -17709.642,E2 -17709.642} C_VEL
LIN {X 0,Y 273.605,Z 729.534,A -85,B 0,C 180,E1 -17711.272,E2 -17711.272} C_VEL
LIN {X 0,Y 272.058,Z 738.787,A -85,B 0,C 180,E1 -17713.07,E2 -17713.07} C_VEL
LIN {X 0,Y 271.153,Z 745.271,A -85,B 0,C 180,E1 -17714.594,E2 -17714.594} C_VEL
LIN {X 0,Y 269.951,Z 753.133,A -85,B 0,C 180,E1 -17716.833,E2 -17716.833} C_VEL
LIN {X 0,Y 269.184,Z 758.486,A -85,B 0,C 180,E1 -17718.708,E2 -17718.708} C_VEL
LIN {X 0,Y 268.659,Z 763.661,A -85,B 0,C 180,E1 -17720.97,E2 -17720.97} C_VEL
LIN {X 0,Y 268.387,Z 767.648,A -85,B 0,C 180,E1 -17723.233,E2 -17723.233} C_VEL
LIN {X 0,Y 268.358,Z 770.56,A -85,B 0,C 180,E1 -17725.494,E2 -17725.494} C_VEL
LIN {X 0,Y 268.371,Z 771.913,A -85,B 0,C 180,E1 -17726.998,E2 -17726.998} C_VEL
LIN {X 0,Y 268.388,Z 772.852,A -85,B 0,C 180,E1 -17728.5,E2 -17728.5} C_VEL
LIN {X 0,Y 268.486,Z 773.388,A -85,B 0,C 180,E1 -17730,E2 -17730} C_VEL
LIN {X 0,Y 268.375,Z 773.472,A -85,B 0,C 180,E1 -17731.501,E2 -17731.501} C_VEL
LIN {X 0,Y 268.339,Z 773.133,A -85,B 0,C 180,E1 -17733.003,E2 -17733.003} C_VEL
LIN {X 0,Y 268.286,Z 771.263,A -85,B 0,C 180,E1 -17736.015,E2 -17736.015} C_VEL
LIN {X 0,Y 268.513,Z 768.742,A -85,B 0,C 180,E1 -17738.277,E2 -17738.277} C_VEL
LIN {X 0,Y 268.992,Z 765.226,A -85,B 0,C 180,E1 -17740.538,E2 -17740.538} C_VEL
LIN {X 0,Y 269.863,Z 760.636,A -85,B 0,C 180,E1 -17742.789,E2 -17742.789} C_VEL
LIN {X 0,Y 271.491,Z 753.754,A -85,B 0,C 180,E1 -17745.387,E2 -17745.387} C_VEL
LIN {X 0,Y 273.1,Z 746.794,A -85,B 0,C 180,E1 -17747.458,E2 -17747.458} C_VEL
LIN {X 0,Y 274.857,Z 738.757,A -85,B 0,C 180,E1 -17749.414,E2 -17749.414} C_VEL
LIN {X 0,Y 277.164,Z 728.703,A -85,B 0,C 180,E1 -17751.377,E2 -17751.377} C_VEL
LIN {X 0,Y 279.318,Z 718.52,A -85,B 0,C 180,E1 -17752.954,E2 -17752.954} C_VEL
LIN {X 0,Y 281.495,Z 707.301,A -85,B 0,C 180,E1 -17754.327,E2 -17754.327} C_VEL
LIN {X 0,Y 283.555,Z 694.816,A -85,B 0,C 180,E1 -17755.508,E2 -17755.508} C_VEL
LIN {X 0,Y 285.284,Z 682.138,A -85,B 0,C 180,E1 -17756.372,E2 -17756.372} C_VEL
LIN {X 0,Y 286.529,Z 669.074,A -85,B 0,C 180,E1 -17756.985,E2 -17756.985} C_VEL
LIN {X 0,Y 288.897,Z 613.235,A -85,B 0,C 180,E1 -17758.55,E2 -17758.55} C_VEL
LIN {X 0,Y 286.269,Z 591.052,A -85,B 0,C 180,E1 -17759.653,E2 -17759.653} C_VEL
LIN {X 0,Y 283.194,Z 574.082,A -85,B 0,C 180,E1 -17760.678,E2 -17760.678} C_VEL
LIN {X 0,Y 277.601,Z 561.847,A -85,B 0,C 180,E1 -17761.982,E2 -17761.982} C_VEL
LIN {X 0,Y 275.731,Z 557.676,A -85,B 0,C 180,E1 -17762.484,E2 -17762.484} C_VEL
LIN {X 0,Y 273.875,Z 549.176,A -85,B 0,C 180,E1 -17765.797,E2 -17765.797} C_VEL
LIN {X 0,Y 271.826,Z 541.407,A -85,B 0,C 180,E1 -17769.136,E2 -17769.136} C_VEL
LIN {X 0,Y 270.216,Z 535.828,A -85,B 0,C 180,E1 -17771.83,E2 -17771.83} C_VEL
LIN {X 0,Y 270.188,Z 535.826,A -85,B 0,C 180,E1 -17775.386,E2 -17775.386} C_VEL
LIN {X 0,Y 270.176,Z 535.83,A -85,B 0,C 180,E1 -17779.434,E2 -17779.434} C_VEL
LIN {X 0,Y 270.252,Z 535.818,A -85,B 0,C 180,E1 -17783.721,E2 -17783.721} C_VEL
LIN {X 0,Y 270.201,Z 535.825,A -85,B 0,C 180,E1 -17786.891,E2 -17786.891} C_VEL
LIN {X 0,Y 270.226,Z 535.824,A -85,B 0,C 180,E1 -17790.386,E2 -17790.386} C_VEL
LIN {X 0,Y 270.26,Z 535.82,A -85,B 0,C 180,E1 -17793.763,E2 -17793.763} C_VEL
LIN {X 0,Y 270.229,Z 535.823,A -85,B 0,C 180,E1 -17797.038,E2 -17797.038} C_VEL
LIN {X 0,Y 270.297,Z 535.812,A -85,B 0,C 180,E1 -17800.243,E2 -17800.243} C_VEL
LIN {X 0,Y 270.398,Z 535.804,A -85,B 0,C 180,E1 -17804.934,E2 -17804.934} C_VEL
LIN {X 0,Y 270.436,Z 535.792,A -85,B 0,C 180,E1 -17809.518,E2 -17809.518} C_VEL
LIN {X 0,Y 270.603,Z 535.777,A -85,B 0,C 180,E1 -17812.538,E2 -17812.538} C_VEL
LIN {X 0,Y 270.782,Z 535.754,A -85,B 0,C 180,E1 -17818.512,E2 -17818.512} C_VEL
LIN {X 0,Y 270.784,Z 535.754,A -85,B 0,C 180,E1 -17821.486,E2 -17821.486} C_VEL
LIN {X 0,Y 270.593,Z 535.779,A -85,B 0,C 180,E1 -17827.461,E2 -17827.461} C_VEL
LIN {X 0,Y 270.406,Z 535.804,A -85,B 0,C 180,E1 -17830.482,E2 -17830.482} C_VEL
LIN {X 0,Y 270.39,Z 535.806,A -85,B 0,C 180,E1 -17835.065,E2 -17835.065} C_VEL
LIN {X 0,Y 270.304,Z 535.934,A -85,B 0,C 180,E1 -17838.67,E2 -17838.67} C_VEL
LIN {X 0,Y 271.469,Z 538.949,A -85,B 0,C 180,E1 -17839.028,E2 -17839.028} C_VEL
LIN {X 0,Y 273.086,Z 541.052,A -85,B 0,C 180,E1 -17839.398,E2 -17839.398} C_VEL
LIN {X 0,Y 280.286,Z 553.123,A -85,B 0,C 180,E1 -17841.048,E2 -17841.048} C_VEL
LIN {X 0,Y 286.158,Z 564.796,A -85,B 0,C 180,E1 -17842.349,E2 -17842.349} C_VEL
LIN {X 0,Y 290.267,Z 574.231,A -85,B 0,C 180,E1 -17843.251,E2 -17843.251} C_VEL
LIN {X 0,Y 287.374,Z 641.334,A -85,B 0,C 180,E1 -17845.13,E2 -17845.13} C_VEL
LIN {X 0,Y 286.306,Z 655.147,A -85,B 0,C 180,E1 -17845.807,E2 -17845.807} C_VEL
LIN {X 0,Y 285.043,Z 667.455,A -85,B 0,C 180,E1 -17846.704,E2 -17846.704} C_VEL
LIN {X 0,Y 283.387,Z 679.285,A -85,B 0,C 180,E1 -17847.862,E2 -17847.862} C_VEL
LIN {X 0,Y 281.64,Z 689.592,A -85,B 0,C 180,E1 -17849.148,E2 -17849.148} C_VEL
LIN {X 0,Y 279.569,Z 699.868,A -85,B 0,C 180,E1 -17850.742,E2 -17850.742} C_VEL
LIN {X 0,Y 277.452,Z 709.328,A -85,B 0,C 180,E1 -17852.588,E2 -17852.588} C_VEL
LIN {X 0,Y 275.39,Z 717.592,A -85,B 0,C 180,E1 -17854.6,E2 -17854.6} C_VEL
LIN {X 0,Y 273.654,Z 724.328,A -85,B 0,C 180,E1 -17856.642,E2 -17856.642} C_VEL
LIN {X 0,Y 271.886,Z 730.865,A -85,B 0,C 180,E1 -17859.154,E2 -17859.154} C_VEL
LIN {X 0,Y 270.774,Z 734.921,A -85,B 0,C 180,E1 -17861.177,E2 -17861.177} C_VEL
LIN {X 0,Y 269.916,Z 738.045,A -85,B 0,C 180,E1 -17863.194,E2 -17863.194} C_VEL
LIN {X 0,Y 269.246,Z 740.338,A -85,B 0,C 180,E1 -17865.191,E2 -17865.191} C_VEL
LIN {X 0,Y 268.757,Z 741.886,A -85,B 0,C 180,E1 -17867.166,E2 -17867.166} C_VEL
LIN {X 0,Y 268.37,Z 742.761,A -85,B 0,C 180,E1 -17869.414,E2 -17869.414} C_VEL
LIN {X 0,Y 268.18,Z 742.705,A -85,B 0,C 180,E1 -17871.829,E2 -17871.829} C_VEL
LIN {X 0,Y 268.273,Z 741.182,A -85,B 0,C 180,E1 -17874.808,E2 -17874.808} C_VEL
LIN {X 0,Y 268.739,Z 738.201,A -85,B 0,C 180,E1 -17877.679,E2 -17877.679} C_VEL
LIN {X 0,Y 269.364,Z 734.067,A -85,B 0,C 180,E1 -17880.283,E2 -17880.283} C_VEL
LIN {X 0,Y 270.296,Z 728.038,A -85,B 0,C 180,E1 -17883.03,E2 -17883.03} C_VEL
LIN {X 0,Y 271.492,Z 720.809,A -85,B 0,C 180,E1 -17885.533,E2 -17885.533} C_VEL
LIN {X 0,Y 272.793,Z 713.013,A -85,B 0,C 180,E1 -17887.657,E2 -17887.657} C_VEL
LIN {X 0,Y 274.367,Z 703.363,A -85,B 0,C 180,E1 -17889.769,E2 -17889.769} C_VEL
LIN {X 0,Y 275.777,Z 693.922,A -85,B 0,C 180,E1 -17891.425,E2 -17891.425} C_VEL
LIN {X 0,Y 277.396,Z 682.181,A -85,B 0,C 180,E1 -17893.062,E2 -17893.062} C_VEL
LIN {X 0,Y 278.776,Z 670.171,A -85,B 0,C 180,E1 -17894.37,E2 -17894.37} C_VEL
LIN {X 0,Y 279.882,Z 658.003,A -85,B 0,C 180,E1 -17895.365,E2 -17895.365} C_VEL
LIN {X 0,Y 280.739,Z 645.05,A -85,B 0,C 180,E1 -17896.125,E2 -17896.125} C_VEL
LIN {X 0,Y 281.287,Z 631.525,A -85,B 0,C 180,E1 -17896.618,E2 -17896.618} C_VEL
LIN {X 0,Y 283.369,Z 568.544,A -85,B 0,C 180,E1 -17898.314,E2 -17898.314} C_VEL
LIN {X 0,Y 282.193,Z 564.476,A -85,B 0,C 180,E1 -17898.533,E2 -17898.533} C_VEL
LIN {X 0,Y 277.293,Z 551.774,A -85,B 0,C 180,E1 -17899.34,E2 -17899.34} C_VEL
LIN {X 0,Y 270.655,Z 536.536,A -85,B 0,C 180,E1 -17900.43,E2 -17900.43} C_VEL
LIN {X 0,Y 270.529,Z 535.791,A -85,B 0,C 180,E1 -17900.467,E2 -17900.467} C_VEL
LIN {X 0,Y 270.538,Z 535.785,A -85,B 0,C 180,E1 -17904.036,E2 -17904.036} C_VEL
LIN {X 0,Y 270.785,Z 535.755,A -85,B 0,C 180,E1 -17908.513,E2 -17908.513} C_VEL
LIN {X 0,Y 270.785,Z 535.754,A -85,B 0,C 180,E1 -17911.487,E2 -17911.487} C_VEL
LIN {X 0,Y 270.608,Z 535.776,A -85,B 0,C 180,E1 -17917.461,E2 -17917.461} C_VEL
LIN {X 0,Y 270.439,Z 535.797,A -85,B 0,C 180,E1 -17920.481,E2 -17920.481} C_VEL
LIN {X 0,Y 270.4,Z 535.804,A -85,B 0,C 180,E1 -17925.064,E2 -17925.064} C_VEL
LIN {X 0,Y 270.298,Z 535.812,A -85,B 0,C 180,E1 -17929.755,E2 -17929.755} C_VEL
LIN {X 0,Y 270.27,Z 535.818,A -85,B 0,C 180,E1 -17934.585,E2 -17934.585} C_VEL
LIN {X 0,Y 270.268,Z 535.817,A -85,B 0,C 180,E1 -17937.908,E2 -17937.908} C_VEL
LIN {X 0,Y 270.18,Z 535.83,A -85,B 0,C 180,E1 -17941.348,E2 -17941.348} C_VEL
LIN {X 0,Y 270.211,Z 535.827,A -85,B 0,C 180,E1 -17944.903,E2 -17944.903} C_VEL
LIN {X 0,Y 270.217,Z 535.822,A -85,B 0,C 180,E1 -17948.717,E2 -17948.717} C_VEL
LIN {X 0,Y 270.251,Z 535.819,A -85,B 0,C 180,E1 -17952.542,E2 -17952.542} C_VEL
LIN {X 0,Y 270.226,Z 535.822,A -85,B 0,C 180,E1 -17956.736,E2 -17956.736} C_VEL
LIN {X 0,Y 270.243,Z 535.819,A -85,B 0,C 180,E1 -17959.448,E2 -17959.448} C_VEL
LIN {X 0,Y 270.25,Z 535.819,A -85,B 0,C 180,E1 -17963.722,E2 -17963.722} C_VEL
LIN {X 0,Y 270.198,Z 535.825,A -85,B 0,C 180,E1 -17966.893,E2 -17966.893} C_VEL
LIN {X 0,Y 270.223,Z 535.819,A -85,B 0,C 180,E1 -17970.387,E2 -17970.387} C_VEL
LIN {X 0,Y 270.257,Z 535.819,A -85,B 0,C 180,E1 -17973.764,E2 -17973.764} C_VEL
LIN {X 0,Y 270.203,Z 535.825,A -85,B 0,C 180,E1 -17977.037,E2 -17977.037} C_VEL
LIN {X 0,Y 270.293,Z 535.807,A -85,B 0,C 180,E1 -17980.245,E2 -17980.245} C_VEL
LIN {X 0,Y 270.39,Z 535.804,A -85,B 0,C 180,E1 -17984.935,E2 -17984.935} C_VEL
LIN {X 0,Y 270.436,Z 535.788,A -85,B 0,C 180,E1 -17989.52,E2 -17989.52} C_VEL
LIN {X 0,Y 270.605,Z 535.771,A -85,B 0,C 180,E1 -17992.539,E2 -17992.539} C_VEL
LIN {X 0,Y 270.537,Z 535.779,A -85,B 0,C 180,E1 -17993.828,E2 -17993.828} C_VEL
LIN {X 0,Y 269.915,Z 535.863,A -85,B 0,C 180,E1 -17995.072,E2 -17995.072} C_VEL
LIN {X 0,Y 267.216,Z 536.199,A -85,B 0,C 180,E1 -17997.103,E2 -17997.103} C_VEL
LIN {X 0,Y 264.106,Z 536.578,A -85,B 0,C 180,E1 -17999.599,E2 -17999.599} C_VEL
LIN {X 0,Y 263.771,Z 536.617,A -85,B 0,C 180,E1 -18000.46,E2 -18000.46} C_VEL
LIN {X 0,Y 263.595,Z 536.647,A -85,B 0,C 180,E1 -18003.057,E2 -18003.057} C_VEL
LIN {X 0,Y 263.553,Z 536.651,A -85,B 0,C 180,E1 -18007.663,E2 -18007.663} C_VEL
LIN {X 0,Y 263.35,Z 536.675,A -85,B 0,C 180,E1 -18010.767,E2 -18010.767} C_VEL
LIN {X 0,Y 263.346,Z 536.68,A -85,B 0,C 180,E1 -18015.479,E2 -18015.479} C_VEL
LIN {X 0,Y 263.26,Z 536.69,A -85,B 0,C 180,E1 -18020.308,E2 -18020.308} C_VEL
LIN {X 0,Y 263.205,Z 536.698,A -85,B 0,C 180,E1 -18025.292,E2 -18025.292} C_VEL
LIN {X 0,Y 263.177,Z 536.701,A -85,B 0,C 180,E1 -18028.731,E2 -18028.731} C_VEL
LIN {X 0,Y 263.131,Z 536.706,A -85,B 0,C 180,E1 -18032.289,E2 -18032.289} C_VEL
LIN {X 0,Y 263.184,Z 536.7,A -85,B 0,C 180,E1 -18035.979,E2 -18035.979} C_VEL
LIN {X 0,Y 263.106,Z 536.709,A -85,B 0,C 180,E1 -18039.873,E2 -18039.873} C_VEL
LIN {X 0,Y 263.137,Z 536.706,A -85,B 0,C 180,E1 -18043.982,E2 -18043.982} C_VEL
LIN {X 0,Y 263.173,Z 536.702,A -85,B 0,C 180,E1 -18048.396,E2 -18048.396} C_VEL
LIN {X 0,Y 263.252,Z 536.886,A -85,B 0,C 180,E1 -18053.048,E2 -18053.048} C_VEL
LIN {X 0,Y 265.747,Z 548.276,A -85,B 0,C 180,E1 -18057.067,E2 -18057.067} C_VEL
LIN {X 0,Y 268.211,Z 560.255,A -85,B 0,C 180,E1 -18061.061,E2 -18061.061} C_VEL
LIN {X 0,Y 268.313,Z 560.836,A -85,B 0,C 180,E1 -18061.21,E2 -18061.21} C_VEL
LIN {X 0,Y 269.841,Z 566.501,A -85,B 0,C 180,E1 -18061.534,E2 -18061.534} C_VEL
LIN {X 0,Y 274.577,Z 602.232,A -85,B 0,C 180,E1 -18063.069,E2 -18063.069} C_VEL
LIN {X 0,Y 275.756,Z 613.388,A -85,B 0,C 180,E1 -18063.507,E2 -18063.507} C_VEL
LIN {X 0,Y 273.916,Z 669.66,A -85,B 0,C 180,E1 -18065.107,E2 -18065.107} C_VEL
LIN {X 0,Y 272.9,Z 683.229,A -85,B 0,C 180,E1 -18065.768,E2 -18065.768} C_VEL
LIN {X 0,Y 271.586,Z 695.625,A -85,B 0,C 180,E1 -18066.657,E2 -18066.657} C_VEL
LIN {X 0,Y 270.046,Z 707.586,A -85,B 0,C 180,E1 -18067.83,E2 -18067.83} C_VEL
LIN {X 0,Y 268.361,Z 719.092,A -85,B 0,C 180,E1 -18069.296,E2 -18069.296} C_VEL
LIN {X 0,Y 266.671,Z 729.488,A -85,B 0,C 180,E1 -18070.966,E2 -18070.966} C_VEL
LIN {X 0,Y 264.968,Z 739.65,A -85,B 0,C 180,E1 -18073.037,E2 -18073.037} C_VEL
LIN {X 0,Y 263.756,Z 747.213,A -85,B 0,C 180,E1 -18074.942,E2 -18074.942} C_VEL
LIN {X 0,Y 262.592,Z 754.625,A -85,B 0,C 180,E1 -18077.244,E2 -18077.244} C_VEL
LIN {X 0,Y 261.95,Z 759.632,A -85,B 0,C 180,E1 -18079.175,E2 -18079.175} C_VEL
LIN {X 0,Y 261.491,Z 764.472,A -85,B 0,C 180,E1 -18081.5,E2 -18081.5} C_VEL
LIN {X 0,Y 261.293,Z 768.147,A -85,B 0,C 180,E1 -18083.824,E2 -18083.824} C_VEL
LIN {X 0,Y 261.265,Z 770.025,A -85,B 0,C 180,E1 -18085.371,E2 -18085.371} C_VEL
LIN {X 0,Y 261.3,Z 771.413,A -85,B 0,C 180,E1 -18086.917,E2 -18086.917} C_VEL
LIN {X 0,Y 261.308,Z 772.376,A -85,B 0,C 180,E1 -18088.459,E2 -18088.459} C_VEL
LIN {X 0,Y 261.398,Z 772.936,A -85,B 0,C 180,E1 -18090,E2 -18090} C_VEL
LIN {X 0,Y 261.294,Z 773.068,A -85,B 0,C 180,E1 -18091.541,E2 -18091.541} C_VEL
LIN {X 0,Y 261.264,Z 772.757,A -85,B 0,C 180,E1 -18093.084,E2 -18093.084} C_VEL
LIN {X 0,Y 261.219,Z 770.933,A -85,B 0,C 180,E1 -18096.178,E2 -18096.178} C_VEL
LIN {X 0,Y 261.337,Z 769.41,A -85,B 0,C 180,E1 -18097.727,E2 -18097.727} C_VEL
LIN {X 0,Y 261.757,Z 766.287,A -85,B 0,C 180,E1 -18100.05,E2 -18100.05} C_VEL
LIN {X 0,Y 262.505,Z 762.12,A -85,B 0,C 180,E1 -18102.367,E2 -18102.367} C_VEL
LIN {X 0,Y 264.088,Z 755.797,A -85,B 0,C 180,E1 -18105.038,E2 -18105.038} C_VEL
LIN {X 0,Y 265.726,Z 749.151,A -85,B 0,C 180,E1 -18107.247,E2 -18107.247} C_VEL
LIN {X 0,Y 267.763,Z 740.512,A -85,B 0,C 180,E1 -18109.551,E2 -18109.551} C_VEL
LIN {X 0,Y 269.869,Z 731.894,A -85,B 0,C 180,E1 -18111.382,E2 -18111.382} C_VEL
LIN {X 0,Y 272.304,Z 721.316,A -85,B 0,C 180,E1 -18113.178,E2 -18113.178} C_VEL
LIN {X 0,Y 274.772,Z 709.485,A -85,B 0,C 180,E1 -18114.76,E2 -18114.76} C_VEL
LIN {X 0,Y 276.885,Z 697.681,A -85,B 0,C 180,E1 -18115.966,E2 -18115.966} C_VEL
LIN {X 0,Y 278.879,Z 684.366,A -85,B 0,C 180,E1 -18116.975,E2 -18116.975} C_VEL
LIN {X 0,Y 280.301,Z 671.74,A -85,B 0,C 180,E1 -18117.635,E2 -18117.635} C_VEL
LIN {X 0,Y 281.23,Z 654.64,A -85,B 0,C 180,E1 -18118.194,E2 -18118.194} C_VEL
LIN {X 0,Y 282.895,Z 613.301,A -85,B 0,C 180,E1 -18119.367,E2 -18119.367} C_VEL
LIN {X 0,Y 280.303,Z 591.13,A -85,B 0,C 180,E1 -18120.511,E2 -18120.511} C_VEL
LIN {X 0,Y 277.716,Z 576.991,A -85,B 0,C 180,E1 -18121.41,E2 -18121.41} C_VEL
LIN {X 0,Y 272.678,Z 565.867,A -85,B 0,C 180,E1 -18122.649,E2 -18122.649} C_VEL
LIN {X 0,Y 268.514,Z 557.175,A -85,B 0,C 180,E1 -18123.733,E2 -18123.733} C_VEL
LIN {X 0,Y 266.51,Z 548.518,A -85,B 0,C 180,E1 -18127.337,E2 -18127.337} C_VEL
LIN {X 0,Y 264.428,Z 541.149,A -85,B 0,C 180,E1 -18130.758,E2 -18130.758} C_VEL
LIN {X 0,Y 263.186,Z 536.698,A -85,B 0,C 180,E1 -18133.037,E2 -18133.037} C_VEL
LIN {X 0,Y 263.138,Z 536.708,A -85,B 0,C 180,E1 -18136.146,E2 -18136.146} C_VEL
LIN {X 0,Y 263.115,Z 536.705,A -85,B 0,C 180,E1 -18140.128,E2 -18140.128} C_VEL
LIN {X 0,Y 263.186,Z 536.7,A -85,B 0,C 180,E1 -18144.021,E2 -18144.021} C_VEL
LIN {X 0,Y 263.131,Z 536.709,A -85,B 0,C 180,E1 -18147.711,E2 -18147.711} C_VEL
LIN {X 0,Y 263.198,Z 536.695,A -85,B 0,C 180,E1 -18151.782,E2 -18151.782} C_VEL
LIN {X 0,Y 263.223,Z 536.69,A -85,B 0,C 180,E1 -18155.199,E2 -18155.199} C_VEL
LIN {X 0,Y 263.259,Z 536.685,A -85,B 0,C 180,E1 -18159.692,E2 -18159.692} C_VEL
LIN {X 0,Y 263.346,Z 536.682,A -85,B 0,C 180,E1 -18164.521,E2 -18164.521} C_VEL
LIN {X 0,Y 263.368,Z 536.674,A -85,B 0,C 180,E1 -18169.233,E2 -18169.233} C_VEL
LIN {X 0,Y 263.565,Z 536.655,A -85,B 0,C 180,E1 -18172.337,E2 -18172.337} C_VEL
LIN {X 0,Y 263.746,Z 536.631,A -85,B 0,C 180,E1 -18178.472,E2 -18178.472} C_VEL
LIN {X 0,Y 263.749,Z 536.63,A -85,B 0,C 180,E1 -18181.526,E2 -18181.526} C_VEL
LIN {X 0,Y 263.553,Z 536.657,A -85,B 0,C 180,E1 -18187.661,E2 -18187.661} C_VEL
LIN {X 0,Y 263.348,Z 536.681,A -85,B 0,C 180,E1 -18190.766,E2 -18190.766} C_VEL
LIN {X 0,Y 263.348,Z 536.681,A -85,B 0,C 180,E1 -18195.477,E2 -18195.477} C_VEL
LIN {X 0,Y 263.262,Z 536.692,A -85,B 0,C 180,E1 -18197.356,E2 -18197.356} C_VEL
LIN {X 0,Y 264.309,Z 539.645,A -85,B 0,C 180,E1 -18197.703,E2 -18197.703} C_VEL
LIN {X 0,Y 266.119,Z 541.849,A -85,B 0,C 180,E1 -18198.146,E2 -18198.146} C_VEL
LIN {X 0,Y 268.198,Z 545.164,A -85,B 0,C 180,E1 -18198.673,E2 -18198.673} C_VEL
LIN {X 0,Y 275.224,Z 556.868,A -85,B 0,C 180,E1 -18200.359,E2 -18200.359} C_VEL
LIN {X 0,Y 280.953,Z 568.4,A -85,B 0,C 180,E1 -18201.705,E2 -18201.705} C_VEL
LIN {X 0,Y 284.401,Z 576.409,A -85,B 0,C 180,E1 -18202.495,E2 -18202.495} C_VEL
LIN {X 0,Y 281.409,Z 642.026,A -85,B 0,C 180,E1 -18204.369,E2 -18204.369} C_VEL
LIN {X 0,Y 280.31,Z 655.618,A -85,B 0,C 180,E1 -18205.054,E2 -18205.054} C_VEL
LIN {X 0,Y 279.001,Z 667.541,A -85,B 0,C 180,E1 -18205.934,E2 -18205.934} C_VEL
LIN {X 0,Y 277.219,Z 679.73,A -85,B 0,C 180,E1 -18207.15,E2 -18207.15} C_VEL
LIN {X 0,Y 275.152,Z 691.159,A -85,B 0,C 180,E1 -18208.622,E2 -18208.622} C_VEL
LIN {X 0,Y 272.814,Z 701.992,A -85,B 0,C 180,E1 -18210.396,E2 -18210.396} C_VEL
LIN {X 0,Y 270.545,Z 711.48,A -85,B 0,C 180,E1 -18212.364,E2 -18212.364} C_VEL
LIN {X 0,Y 268.435,Z 719.432,A -85,B 0,C 180,E1 -18214.418,E2 -18214.418} C_VEL
LIN {X 0,Y 266.651,Z 725.893,A -85,B 0,C 180,E1 -18216.501,E2 -18216.501} C_VEL
LIN {X 0,Y 264.847,Z 732.14,A -85,B 0,C 180,E1 -18219.09,E2 -18219.09} C_VEL
LIN {X 0,Y 263.366,Z 737.095,A -85,B 0,C 180,E1 -18221.845,E2 -18221.845} C_VEL
LIN {X 0,Y 262.518,Z 739.989,A -85,B 0,C 180,E1 -18224.111,E2 -18224.111} C_VEL
LIN {X 0,Y 261.827,Z 741.997,A -85,B 0,C 180,E1 -18226.446,E2 -18226.446} C_VEL
LIN {X 0,Y 261.366,Z 743.079,A -85,B 0,C 180,E1 -18228.842,E2 -18228.842} C_VEL
LIN {X 0,Y 261.096,Z 743.114,A -85,B 0,C 180,E1 -18231.751,E2 -18231.751} C_VEL
LIN {X 0,Y 261.137,Z 742.218,A -85,B 0,C 180,E1 -18233.841,E2 -18233.841} C_VEL
LIN {X 0,Y 261.395,Z 740.075,A -85,B 0,C 180,E1 -18236.456,E2 -18236.456} C_VEL
LIN {X 0,Y 262.005,Z 736.218,A -85,B 0,C 180,E1 -18239.36,E2 -18239.36} C_VEL
LIN {X 0,Y 262.78,Z 731.331,A -85,B 0,C 180,E1 -18241.953,E2 -18241.953} C_VEL
LIN {X 0,Y 263.771,Z 725.451,A -85,B 0,C 180,E1 -18244.344,E2 -18244.344} C_VEL
LIN {X 0,Y 264.97,Z 718.602,A -85,B 0,C 180,E1 -18246.556,E2 -18246.556} C_VEL
LIN {X 0,Y 266.44,Z 710.138,A -85,B 0,C 180,E1 -18248.735,E2 -18248.735} C_VEL
LIN {X 0,Y 268.011,Z 700.477,A -85,B 0,C 180,E1 -18250.736,E2 -18250.736} C_VEL
LIN {X 0,Y 269.484,Z 690.807,A -85,B 0,C 180,E1 -18252.352,E2 -18252.352} C_VEL
LIN {X 0,Y 271.023,Z 679.421,A -85,B 0,C 180,E1 -18253.866,E2 -18253.866} C_VEL
LIN {X 0,Y 272.419,Z 667.014,A -85,B 0,C 180,E1 -18255.145,E2 -18255.145} C_VEL
LIN {X 0,Y 273.425,Z 655.299,A -85,B 0,C 180,E1 -18256.057,E2 -18256.057} C_VEL
LIN {X 0,Y 274.236,Z 642.508,A -85,B 0,C 180,E1 -18256.748,E2 -18256.748} C_VEL
LIN {X 0,Y 274.877,Z 625.778,A -85,B 0,C 180,E1 -18257.287,E2 -18257.287} C_VEL
LIN {X 0,Y 276.676,Z 569.101,A -85,B 0,C 180,E1 -18258.863,E2 -18258.863} C_VEL
LIN {X 0,Y 271.563,Z 555.514,A -85,B 0,C 180,E1 -18259.742,E2 -18259.742} C_VEL
LIN {X 0,Y 263.631,Z 537.339,A -85,B 0,C 180,E1 -18261.088,E2 -18261.088} C_VEL
LIN {X 0,Y 263.512,Z 536.665,A -85,B 0,C 180,E1 -18261.144,E2 -18261.144} C_VEL
LIN {X 0,Y 263.509,Z 536.66,A -85,B 0,C 180,E1 -18263.876,E2 -18263.876} C_VEL
LIN {X 0,Y 263.749,Z 536.631,A -85,B 0,C 180,E1 -18268.473,E2 -18268.473} C_VEL
LIN {X 0,Y 263.749,Z 536.631,A -85,B 0,C 180,E1 -18271.527,E2 -18271.527} C_VEL
LIN {X 0,Y 263.57,Z 536.652,A -85,B 0,C 180,E1 -18277.661,E2 -18277.661} C_VEL
LIN {X 0,Y 263.371,Z 536.679,A -85,B 0,C 180,E1 -18280.765,E2 -18280.765} C_VEL
LIN {X 0,Y 263.348,Z 536.679,A -85,B 0,C 180,E1 -18285.478,E2 -18285.478} C_VEL
LIN {X 0,Y 263.26,Z 536.688,A -85,B 0,C 180,E1 -18290.306,E2 -18290.306} C_VEL
LIN {X 0,Y 263.205,Z 536.698,A -85,B 0,C 180,E1 -18295.291,E2 -18295.291} C_VEL
LIN {X 0,Y 263.176,Z 536.703,A -85,B 0,C 180,E1 -18298.729,E2 -18298.729} C_VEL
LIN {X 0,Y 263.13,Z 536.706,A -85,B 0,C 180,E1 -18302.288,E2 -18302.288} C_VEL
LIN {X 0,Y 263.185,Z 536.699,A -85,B 0,C 180,E1 -18305.977,E2 -18305.977} C_VEL
LIN {X 0,Y 263.157,Z 536.699,A -85,B 0,C 180,E1 -18309.862,E2 -18309.862} C_VEL
LIN {X 0,Y 263.186,Z 536.699,A -85,B 0,C 180,E1 -18313.864,E2 -18313.864} C_VEL
LIN {X 0,Y 263.206,Z 536.689,A -85,B 0,C 180,E1 -18318.385,E2 -18318.385} C_VEL
LIN {X 0,Y 263.198,Z 536.7,A -85,B 0,C 180,E1 -18323.23,E2 -18323.23} C_VEL
LIN {X 0,Y 263.178,Z 536.696,A -85,B 0,C 180,E1 -18325.89,E2 -18325.89} C_VEL
LIN {X 0,Y 263.145,Z 536.702,A -85,B 0,C 180,E1 -18329.507,E2 -18329.507} C_VEL
LIN {X 0,Y 263.187,Z 536.702,A -85,B 0,C 180,E1 -18333.003,E2 -18333.003} C_VEL
LIN {X 0,Y 263.148,Z 536.702,A -85,B 0,C 180,E1 -18336.385,E2 -18336.385} C_VEL
LIN {X 0,Y 263.256,Z 536.684,A -85,B 0,C 180,E1 -18339.694,E2 -18339.694} C_VEL
LIN {X 0,Y 263.338,Z 536.68,A -85,B 0,C 180,E1 -18344.522,E2 -18344.522} C_VEL
LIN {X 0,Y 263.368,Z 536.671,A -85,B 0,C 180,E1 -18349.235,E2 -18349.235} C_VEL
LIN {X 0,Y 263.567,Z 536.646,A -85,B 0,C 180,E1 -18352.339,E2 -18352.339} C_VEL
LIN {X 0,Y 263.746,Z 536.625,A -85,B 0,C 180,E1 -18358.474,E2 -18358.474} C_VEL
LIN {X 0,Y 263.771,Z 536.617,A -85,B 0,C 180,E1 -18360.46,E2 -18360.46} C_VEL
LIN {X 0,Y 263.029,Z 536.715,A -85,B 0,C 180,E1 -18361.731,E2 -18361.731} C_VEL
LIN {X 0,Y 260.055,Z 537.088,A -85,B 0,C 180,E1 -18363.799,E2 -18363.799} C_VEL
LIN {X 0,Y 257.578,Z 537.399,A -85,B 0,C 180,E1 -18365.482,E2 -18365.482} C_VEL
LIN {X 0,Y 256.544,Z 537.526,A -85,B 0,C 180,E1 -18366.789,E2 -18366.789} C_VEL
LIN {X 0,Y 256.474,Z 537.529,A -85,B 0,C 180,E1 -18367.232,E2 -18367.232} C_VEL
LIN {X 0,Y 256.292,Z 537.556,A -85,B 0,C 180,E1 -18371.068,E2 -18371.068} C_VEL
LIN {X 0,Y 256.295,Z 537.555,A -85,B 0,C 180,E1 -18375.916,E2 -18375.916} C_VEL
LIN {X 0,Y 256.163,Z 537.576,A -85,B 0,C 180,E1 -18380.896,E2 -18380.896} C_VEL
LIN {X 0,Y 256.185,Z 537.571,A -85,B 0,C 180,E1 -18385.14,E2 -18385.14} C_VEL
LIN {X 0,Y 256.111,Z 537.581,A -85,B 0,C 180,E1 -18389.601,E2 -18389.601} C_VEL
LIN {X 0,Y 256.083,Z 537.586,A -85,B 0,C 180,E1 -18393.291,E2 -18393.291} C_VEL
LIN {X 0,Y 256.125,Z 537.581,A -85,B 0,C 180,E1 -18397.276,E2 -18397.276} C_VEL
LIN {X 0,Y 256.078,Z 537.585,A -85,B 0,C 180,E1 -18402.184,E2 -18402.184} C_VEL
LIN {X 0,Y 256.103,Z 537.583,A -85,B 0,C 180,E1 -18406.683,E2 -18406.683} C_VEL
LIN {X 0,Y 256.11,Z 537.585,A -85,B 0,C 180,E1 -18410.866,E2 -18410.866} C_VEL
LIN {X 0,Y 256.173,Z 537.658,A -85,B 0,C 180,E1 -18412.482,E2 -18412.482} C_VEL
LIN {X 0,Y 258.373,Z 547.588,A -85,B 0,C 180,E1 -18416.11,E2 -18416.11} C_VEL
LIN {X 0,Y 260.989,Z 560.148,A -85,B 0,C 180,E1 -18420.449,E2 -18420.449} C_VEL
LIN {X 0,Y 263.343,Z 567.531,A -85,B 0,C 180,E1 -18420.955,E2 -18420.955} C_VEL
LIN {X 0,Y 268.314,Z 605.717,A -85,B 0,C 180,E1 -18422.643,E2 -18422.643} C_VEL
LIN {X 0,Y 269.167,Z 613.533,A -85,B 0,C 180,E1 -18422.961,E2 -18422.961} C_VEL
LIN {X 0,Y 267.248,Z 669.56,A -85,B 0,C 180,E1 -18424.598,E2 -18424.598} C_VEL
LIN {X 0,Y 266.212,Z 683.028,A -85,B 0,C 180,E1 -18425.275,E2 -18425.275} C_VEL
LIN {X 0,Y 264.789,Z 695.893,A -85,B 0,C 180,E1 -18426.228,E2 -18426.228} C_VEL
LIN {X 0,Y 263.211,Z 707.685,A -85,B 0,C 180,E1 -18427.43,E2 -18427.43} C_VEL
LIN {X 0,Y 261.483,Z 719.102,A -85,B 0,C 180,E1 -18428.932,E2 -18428.932} C_VEL
LIN {X 0,Y 259.746,Z 729.413,A -85,B 0,C 180,E1 -18430.644,E2 -18430.644} C_VEL
LIN {X 0,Y 258.051,Z 738.673,A -85,B 0,C 180,E1 -18432.568,E2 -18432.568} C_VEL
LIN {X 0,Y 257.138,Z 744.96,A -85,B 0,C 180,E1 -18434.139,E2 -18434.139} C_VEL
LIN {X 0,Y 255.855,Z 752.707,A -85,B 0,C 180,E1 -18436.498,E2 -18436.498} C_VEL
LIN {X 0,Y 254.94,Z 758.917,A -85,B 0,C 180,E1 -18438.874,E2 -18438.874} C_VEL
LIN {X 0,Y 254.436,Z 763.823,A -85,B 0,C 180,E1 -18441.262,E2 -18441.262} C_VEL
LIN {X 0,Y 254.228,Z 767.561,A -85,B 0,C 180,E1 -18443.652,E2 -18443.652} C_VEL
LIN {X 0,Y 254.18,Z 769.472,A -85,B 0,C 180,E1 -18445.242,E2 -18445.242} C_VEL
LIN {X 0,Y 254.229,Z 770.911,A -85,B 0,C 180,E1 -18446.831,E2 -18446.831} C_VEL
LIN {X 0,Y 254.229,Z 771.9,A -85,B 0,C 180,E1 -18448.416,E2 -18448.416} C_VEL
LIN {X 0,Y 254.313,Z 772.485,A -85,B 0,C 180,E1 -18450,E2 -18450} C_VEL
LIN {X 0,Y 254.215,Z 772.653,A -85,B 0,C 180,E1 -18451.584,E2 -18451.584} C_VEL
LIN {X 0,Y 254.167,Z 772.379,A -85,B 0,C 180,E1 -18453.17,E2 -18453.17} C_VEL
LIN {X 0,Y 254.149,Z 770.603,A -85,B 0,C 180,E1 -18456.35,E2 -18456.35} C_VEL
LIN {X 0,Y 254.267,Z 769.12,A -85,B 0,C 180,E1 -18457.944,E2 -18457.944} C_VEL
LIN {X 0,Y 254.731,Z 766.051,A -85,B 0,C 180,E1 -18460.331,E2 -18460.331} C_VEL
LIN {X 0,Y 255.535,Z 761.952,A -85,B 0,C 180,E1 -18462.71,E2 -18462.71} C_VEL
LIN {X 0,Y 257.216,Z 755.727,A -85,B 0,C 180,E1 -18465.45,E2 -18465.45} C_VEL
LIN {X 0,Y 258.648,Z 750.211,A -85,B 0,C 180,E1 -18467.391,E2 -18467.391} C_VEL
LIN {X 0,Y 260.691,Z 742.11,A -85,B 0,C 180,E1 -18469.693,E2 -18469.693} C_VEL
LIN {X 0,Y 263.268,Z 732.114,A -85,B 0,C 180,E1 -18471.945,E2 -18471.945} C_VEL
LIN {X 0,Y 265.82,Z 721.742,A -85,B 0,C 180,E1 -18473.777,E2 -18473.777} C_VEL
LIN {X 0,Y 268.385,Z 710.139,A -85,B 0,C 180,E1 -18475.391,E2 -18475.391} C_VEL
LIN {X 0,Y 270.587,Z 698.769,A -85,B 0,C 180,E1 -18476.617,E2 -18476.617} C_VEL
LIN {X 0,Y 272.637,Z 685.919,A -85,B 0,C 180,E1 -18477.645,E2 -18477.645} C_VEL
LIN {X 0,Y 274.283,Z 672.441,A -85,B 0,C 180,E1 -18478.4,E2 -18478.4} C_VEL
LIN {X 0,Y 275.199,Z 657.629,A -85,B 0,C 180,E1 -18478.922,E2 -18478.922} C_VEL
LIN {X 0,Y 277.065,Z 614.216,A -85,B 0,C 180,E1 -18480.174,E2 -18480.174} C_VEL
LIN {X 0,Y 274.575,Z 592.538,A -85,B 0,C 180,E1 -18481.341,E2 -18481.341} C_VEL
LIN {X 0,Y 272.354,Z 579.946,A -85,B 0,C 180,E1 -18482.174,E2 -18482.174} C_VEL
LIN {X 0,Y 266.101,Z 566.231,A -85,B 0,C 180,E1 -18483.796,E2 -18483.796} C_VEL
LIN {X 0,Y 262.979,Z 560.307,A -85,B 0,C 180,E1 -18484.627,E2 -18484.627} C_VEL
LIN {X 0,Y 261.212,Z 556.505,A -85,B 0,C 180,E1 -18485.173,E2 -18485.173} C_VEL
LIN {X 0,Y 259.414,Z 548.898,A -85,B 0,C 180,E1 -18488.543,E2 -18488.543} C_VEL
LIN {X 0,Y 257.146,Z 541.074,A -85,B 0,C 180,E1 -18492.444,E2 -18492.444} C_VEL
LIN {X 0,Y 256.077,Z 537.587,A -85,B 0,C 180,E1 -18494.425,E2 -18494.425} C_VEL
LIN {X 0,Y 256.06,Z 537.589,A -85,B 0,C 180,E1 -18498.797,E2 -18498.797} C_VEL
LIN {X 0,Y 256.143,Z 537.573,A -85,B 0,C 180,E1 -18502.869,E2 -18502.869} C_VEL
LIN {X 0,Y 256.083,Z 537.582,A -85,B 0,C 180,E1 -18506.709,E2 -18506.709} C_VEL
LIN {X 0,Y 256.135,Z 537.577,A -85,B 0,C 180,E1 -18511.404,E2 -18511.404} C_VEL
LIN {X 0,Y 256.163,Z 537.567,A -85,B 0,C 180,E1 -18515.698,E2 -18515.698} C_VEL
LIN {X 0,Y 256.162,Z 537.568,A -85,B 0,C 180,E1 -18519.104,E2 -18519.104} C_VEL
LIN {X 0,Y 256.295,Z 537.558,A -85,B 0,C 180,E1 -18524.084,E2 -18524.084} C_VEL
LIN {X 0,Y 256.304,Z 537.557,A -85,B 0,C 180,E1 -18528.933,E2 -18528.933} C_VEL
LIN {X 0,Y 256.533,Z 537.53,A -85,B 0,C 180,E1 -18532.126,E2 -18532.126} C_VEL
LIN {X 0,Y 256.709,Z 537.507,A -85,B 0,C 180,E1 -18538.43,E2 -18538.43} C_VEL
LIN {X 0,Y 256.712,Z 537.507,A -85,B 0,C 180,E1 -18541.568,E2 -18541.568} C_VEL
LIN {X 0,Y 256.466,Z 537.533,A -85,B 0,C 180,E1 -18546.72,E2 -18546.72} C_VEL
LIN {X 0,Y 256.421,Z 537.541,A -85,B 0,C 180,E1 -18549.464,E2 -18549.464} C_VEL
LIN {X 0,Y 256.247,Z 537.566,A -85,B 0,C 180,E1 -18554.29,E2 -18554.29} C_VEL
LIN {X 0,Y 256.339,Z 537.727,A -85,B 0,C 180,E1 -18555.955,E2 -18555.955} C_VEL
LIN {X 0,Y 257.322,Z 540.475,A -85,B 0,C 180,E1 -18556.294,E2 -18556.294} C_VEL
LIN {X 0,Y 259.228,Z 542.879,A -85,B 0,C 180,E1 -18556.805,E2 -18556.805} C_VEL
LIN {X 0,Y 261.411,Z 546.29,A -85,B 0,C 180,E1 -18557.402,E2 -18557.402} C_VEL
LIN {X 0,Y 267.361,Z 555.835,A -85,B 0,C 180,E1 -18558.944,E2 -18558.944} C_VEL
LIN {X 0,Y 272.402,Z 564.875,A -85,B 0,C 180,E1 -18560.186,E2 -18560.186} C_VEL
LIN {X 0,Y 278.359,Z 577.932,A -85,B 0,C 180,E1 -18561.644,E2 -18561.644} C_VEL
LIN {X 0,Y 278.516,Z 580.258,A -85,B 0,C 180,E1 -18561.753,E2 -18561.753} C_VEL
LIN {X 0,Y 275.491,Z 642.779,A -85,B 0,C 180,E1 -18563.578,E2 -18563.578} C_VEL
LIN {X 0,Y 274.283,Z 656.675,A -85,B 0,C 180,E1 -18564.296,E2 -18564.296} C_VEL
LIN {X 0,Y 272.775,Z 669.556,A -85,B 0,C 180,E1 -18565.301,E2 -18565.301} C_VEL
LIN {X 0,Y 270.81,Z 681.899,A -85,B 0,C 180,E1 -18566.593,E2 -18566.593} C_VEL
LIN {X 0,Y 268.698,Z 692.904,A -85,B 0,C 180,E1 -18568.086,E2 -18568.086} C_VEL
LIN {X 0,Y 266.4,Z 702.809,A -85,B 0,C 180,E1 -18569.776,E2 -18569.776} C_VEL
LIN {X 0,Y 264.176,Z 711.617,A -85,B 0,C 180,E1 -18571.648,E2 -18571.648} C_VEL
LIN {X 0,Y 261.947,Z 719.534,A -85,B 0,C 180,E1 -18573.726,E2 -18573.726} C_VEL
LIN {X 0,Y 260.081,Z 726.003,A -85,B 0,C 180,E1 -18575.84,E2 -18575.84} C_VEL
LIN {X 0,Y 258.47,Z 731.205,A -85,B 0,C 180,E1 -18577.953,E2 -18577.953} C_VEL
LIN {X 0,Y 257.166,Z 735.358,A -85,B 0,C 180,E1 -18580.077,E2 -18580.077} C_VEL
LIN {X 0,Y 256.149,Z 738.586,A -85,B 0,C 180,E1 -18582.202,E2 -18582.202} C_VEL
LIN {X 0,Y 255.36,Z 740.981,A -85,B 0,C 180,E1 -18584.311,E2 -18584.311} C_VEL
LIN {X 0,Y 254.751,Z 742.585,A -85,B 0,C 180,E1 -18586.396,E2 -18586.396} C_VEL
LIN {X 0,Y 254.344,Z 743.46,A -85,B 0,C 180,E1 -18588.46,E2 -18588.46} C_VEL
LIN {X 0,Y 254.064,Z 743.657,A -85,B 0,C 180,E1 -18590.762,E2 -18590.762} C_VEL
LIN {X 0,Y 254.013,Z 742.859,A -85,B 0,C 180,E1 -18593.356,E2 -18593.356} C_VEL
LIN {X 0,Y 254.316,Z 740.492,A -85,B 0,C 180,E1 -18596.449,E2 -18596.449} C_VEL
LIN {X 0,Y 254.791,Z 737.63,A -85,B 0,C 180,E1 -18598.767,E2 -18598.767} C_VEL
LIN {X 0,Y 255.404,Z 733.886,A -85,B 0,C 180,E1 -18601.023,E2 -18601.023} C_VEL
LIN {X 0,Y 256.319,Z 728.466,A -85,B 0,C 180,E1 -18603.542,E2 -18603.542} C_VEL
LIN {X 0,Y 257.65,Z 720.78,A -85,B 0,C 180,E1 -18606.276,E2 -18606.276} C_VEL
LIN {X 0,Y 259.084,Z 712.771,A -85,B 0,C 180,E1 -18608.519,E2 -18608.519} C_VEL
LIN {X 0,Y 260.728,Z 703.343,A -85,B 0,C 180,E1 -18610.634,E2 -18610.634} C_VEL
LIN {X 0,Y 262.346,Z 693.137,A -85,B 0,C 180,E1 -18612.46,E2 -18612.46} C_VEL
LIN {X 0,Y 264.064,Z 681.308,A -85,B 0,C 180,E1 -18614.14,E2 -18614.14} C_VEL
LIN {X 0,Y 265.457,Z 669.487,A -85,B 0,C 180,E1 -18615.433,E2 -18615.433} C_VEL
LIN {X 0,Y 266.721,Z 656.045,A -85,B 0,C 180,E1 -18616.534,E2 -18616.534} C_VEL
LIN {X 0,Y 267.568,Z 643.21,A -85,B 0,C 180,E1 -18617.254,E2 -18617.254} C_VEL
LIN {X 0,Y 268.218,Z 627.351,A -85,B 0,C 180,E1 -18617.785,E2 -18617.785} C_VEL
LIN {X 0,Y 270.126,Z 570.8,A -85,B 0,C 180,E1 -18619.392,E2 -18619.392} C_VEL
LIN {X 0,Y 265.461,Z 558.372,A -85,B 0,C 180,E1 -18620.226,E2 -18620.226} C_VEL
LIN {X 0,Y 256.626,Z 538.26,A -85,B 0,C 180,E1 -18621.768,E2 -18621.768} C_VEL
LIN {X 0,Y 256.495,Z 537.537,A -85,B 0,C 180,E1 -18621.844,E2 -18621.844} C_VEL
LIN {X 0,Y 256.336,Z 537.555,A -85,B 0,C 180,E1 -18625.282,E2 -18625.282} C_VEL
LIN {X 0,Y 256.712,Z 537.508,A -85,B 0,C 180,E1 -18628.431,E2 -18628.431} C_VEL
LIN {X 0,Y 256.712,Z 537.507,A -85,B 0,C 180,E1 -18631.569,E2 -18631.569} C_VEL
LIN {X 0,Y 256.537,Z 537.527,A -85,B 0,C 180,E1 -18637.873,E2 -18637.873} C_VEL
LIN {X 0,Y 256.307,Z 537.558,A -85,B 0,C 180,E1 -18641.066,E2 -18641.066} C_VEL
LIN {X 0,Y 256.297,Z 537.556,A -85,B 0,C 180,E1 -18645.915,E2 -18645.915} C_VEL
LIN {X 0,Y 256.164,Z 537.576,A -85,B 0,C 180,E1 -18650.895,E2 -18650.895} C_VEL
LIN {X 0,Y 256.185,Z 537.573,A -85,B 0,C 180,E1 -18655.138,E2 -18655.138} C_VEL
LIN {X 0,Y 256.11,Z 537.581,A -85,B 0,C 180,E1 -18659.599,E2 -18659.599} C_VEL
LIN {X 0,Y 256.081,Z 537.586,A -85,B 0,C 180,E1 -18663.29,E2 -18663.29} C_VEL
LIN {X 0,Y 256.137,Z 537.576,A -85,B 0,C 180,E1 -18667.278,E2 -18667.278} C_VEL
LIN {X 0,Y 256.128,Z 537.58,A -85,B 0,C 180,E1 -18671.188,E2 -18671.188} C_VEL
LIN {X 0,Y 256.111,Z 537.579,A -85,B 0,C 180,E1 -18675.517,E2 -18675.517} C_VEL
LIN {X 0,Y 256.126,Z 537.572,A -85,B 0,C 180,E1 -18678.812,E2 -18678.812} C_VEL
LIN {X 0,Y 256.148,Z 537.578,A -85,B 0,C 180,E1 -18682.871,E2 -18682.871} C_VEL
LIN {X 0,Y 256.079,Z 537.582,A -85,B 0,C 180,E1 -18686.71,E2 -18686.71} C_VEL
LIN {X 0,Y 256.133,Z 537.579,A -85,B 0,C 180,E1 -18691.405,E2 -18691.405} C_VEL
LIN {X 0,Y 256.136,Z 537.576,A -85,B 0,C 180,E1 -18695.697,E2 -18695.697} C_VEL
LIN {X 0,Y 256.155,Z 537.569,A -85,B 0,C 180,E1 -18699.105,E2 -18699.105} C_VEL
LIN {X 0,Y 256.288,Z 537.557,A -85,B 0,C 180,E1 -18704.085,E2 -18704.085} C_VEL
LIN {X 0,Y 256.304,Z 537.553,A -85,B 0,C 180,E1 -18708.935,E2 -18708.935} C_VEL
LIN {X 0,Y 256.534,Z 537.522,A -85,B 0,C 180,E1 -18712.128,E2 -18712.128} C_VEL
LIN {X 0,Y 256.709,Z 537.502,A -85,B 0,C 180,E1 -18718.432,E2 -18718.432} C_VEL
LIN {X 0,Y 256.717,Z 537.502,A -85,B 0,C 180,E1 -18721.57,E2 -18721.57} C_VEL
LIN {X 0,Y 256.474,Z 537.529,A -85,B 0,C 180,E1 -18727.232,E2 -18727.232} C_VEL
LIN {X 0,Y 256.171,Z 537.568,A -85,B 0,C 180,E1 -18728.108,E2 -18728.108} C_VEL
LIN {X 0,Y 254.796,Z 537.742,A -85,B 0,C 180,E1 -18729.399,E2 -18729.399} C_VEL
LIN {X 0,Y 250.333,Z 538.299,A -85,B 0,C 180,E1 -18732.406,E2 -18732.406} C_VEL
LIN {X 0,Y 249.263,Z 538.434,A -85,B 0,C 180,E1 -18733.754,E2 -18733.754} C_VEL
LIN {X 0,Y 249.184,Z 538.442,A -85,B 0,C 180,E1 -18734.212,E2 -18734.212} C_VEL
LIN {X 0,Y 249.214,Z 538.437,A -85,B 0,C 180,E1 -18736.504,E2 -18736.504} C_VEL
LIN {X 0,Y 249.084,Z 538.458,A -85,B 0,C 180,E1 -18741.519,E2 -18741.519} C_VEL
LIN {X 0,Y 249.128,Z 538.453,A -85,B 0,C 180,E1 -18745.483,E2 -18745.483} C_VEL
LIN {X 0,Y 249.081,Z 538.458,A -85,B 0,C 180,E1 -18748.994,E2 -18748.994} C_VEL
LIN {X 0,Y 249.034,Z 538.463,A -85,B 0,C 180,E1 -18752.426,E2 -18752.426} C_VEL
LIN {X 0,Y 249.066,Z 538.458,A -85,B 0,C 180,E1 -18756.34,E2 -18756.34} C_VEL
LIN {X 0,Y 249.006,Z 538.465,A -85,B 0,C 180,E1 -18760.479,E2 -18760.479} C_VEL
LIN {X 0,Y 249.018,Z 538.466,A -85,B 0,C 180,E1 -18764.877,E2 -18764.877} C_VEL
LIN {X 0,Y 249.062,Z 538.463,A -85,B 0,C 180,E1 -18767.374,E2 -18767.374} C_VEL
LIN {X 0,Y 249.127,Z 538.543,A -85,B 0,C 180,E1 -18771.935,E2 -18771.935} C_VEL
LIN {X 0,Y 251.527,Z 549.418,A -85,B 0,C 180,E1 -18776.026,E2 -18776.026} C_VEL
LIN {X 0,Y 253.704,Z 559.913,A -85,B 0,C 180,E1 -18779.743,E2 -18779.743} C_VEL
LIN {X 0,Y 257.052,Z 569.905,A -85,B 0,C 180,E1 -18780.422,E2 -18780.422} C_VEL
LIN {X 0,Y 261.911,Z 608.041,A -85,B 0,C 180,E1 -18782.144,E2 -18782.144} C_VEL
LIN {X 0,Y 262.566,Z 614.688,A -85,B 0,C 180,E1 -18782.419,E2 -18782.419} C_VEL
LIN {X 0,Y 260.589,Z 669.658,A -85,B 0,C 180,E1 -18784.072,E2 -18784.072} C_VEL
LIN {X 0,Y 259.511,Z 682.813,A -85,B 0,C 180,E1 -18784.753,E2 -18784.753} C_VEL
LIN {X 0,Y 258.153,Z 695.11,A -85,B 0,C 180,E1 -18785.685,E2 -18785.685} C_VEL
LIN {X 0,Y 256.653,Z 706.203,A -85,B 0,C 180,E1 -18786.82,E2 -18786.82} C_VEL
LIN {X 0,Y 254.804,Z 717.806,A -85,B 0,C 180,E1 -18788.352,E2 -18788.352} C_VEL
LIN {X 0,Y 252.989,Z 728.29,A -85,B 0,C 180,E1 -18790.105,E2 -18790.105} C_VEL
LIN {X 0,Y 251.271,Z 737.713,A -85,B 0,C 180,E1 -18792.082,E2 -18792.082} C_VEL
LIN {X 0,Y 249.984,Z 745.474,A -85,B 0,C 180,E1 -18794.091,E2 -18794.091} C_VEL
LIN {X 0,Y 248.696,Z 753.053,A -85,B 0,C 180,E1 -18796.518,E2 -18796.518} C_VEL
LIN {X 0,Y 247.708,Z 760.02,A -85,B 0,C 180,E1 -18799.373,E2 -18799.373} C_VEL
LIN {X 0,Y 247.267,Z 764.582,A -85,B 0,C 180,E1 -18801.83,E2 -18801.83} C_VEL
LIN {X 0,Y 247.167,Z 768.131,A -85,B 0,C 180,E1 -18804.391,E2 -18804.391} C_VEL
LIN {X 0,Y 247.159,Z 770.408,A -85,B 0,C 180,E1 -18806.74,E2 -18806.74} C_VEL
LIN {X 0,Y 247.153,Z 771.422,A -85,B 0,C 180,E1 -18808.371,E2 -18808.371} C_VEL
LIN {X 0,Y 247.23,Z 772.032,A -85,B 0,C 180,E1 -18810,E2 -18810} C_VEL
LIN {X 0,Y 247.137,Z 772.227,A -85,B 0,C 180,E1 -18811.63,E2 -18811.63} C_VEL
LIN {X 0,Y 247.072,Z 772.004,A -85,B 0,C 180,E1 -18813.261,E2 -18813.261} C_VEL
LIN {X 0,Y 247.059,Z 770.287,A -85,B 0,C 180,E1 -18816.533,E2 -18816.533} C_VEL
LIN {X 0,Y 247.2,Z 768.832,A -85,B 0,C 180,E1 -18818.172,E2 -18818.172} C_VEL
LIN {X 0,Y 247.722,Z 765.82,A -85,B 0,C 180,E1 -18820.626,E2 -18820.626} C_VEL
LIN {X 0,Y 248.577,Z 761.782,A -85,B 0,C 180,E1 -18823.072,E2 -18823.072} C_VEL
LIN {X 0,Y 250.355,Z 755.657,A -85,B 0,C 180,E1 -18825.884,E2 -18825.884} C_VEL
LIN {X 0,Y 252.289,Z 748.83,A -85,B 0,C 180,E1 -18828.313,E2 -18828.313} C_VEL
LIN {X 0,Y 254.421,Z 740.748,A -85,B 0,C 180,E1 -18830.621,E2 -18830.621} C_VEL
LIN {X 0,Y 256.701,Z 732.394,A -85,B 0,C 180,E1 -18832.537,E2 -18832.537} C_VEL
LIN {X 0,Y 259.363,Z 722.235,A -85,B 0,C 180,E1 -18834.407,E2 -18834.407} C_VEL
LIN {X 0,Y 262.025,Z 710.822,A -85,B 0,C 180,E1 -18836.053,E2 -18836.053} C_VEL
LIN {X 0,Y 264.297,Z 699.723,A -85,B 0,C 180,E1 -18837.303,E2 -18837.303} C_VEL
LIN {X 0,Y 266.379,Z 687.484,A -85,B 0,C 180,E1 -18838.352,E2 -18838.352} C_VEL
LIN {X 0,Y 268.227,Z 673.882,A -85,B 0,C 180,E1 -18839.155,E2 -18839.155} C_VEL
LIN {X 0,Y 269.251,Z 660.667,A -85,B 0,C 180,E1 -18839.677,E2 -18839.677} C_VEL
LIN {X 0,Y 271.317,Z 614.571,A -85,B 0,C 180,E1 -18841.049,E2 -18841.049} C_VEL
LIN {X 0,Y 268.893,Z 593.483,A -85,B 0,C 180,E1 -18842.242,E2 -18842.242} C_VEL
LIN {X 0,Y 267,Z 582.835,A -85,B 0,C 180,E1 -18842.979,E2 -18842.979} C_VEL
LIN {X 0,Y 261.162,Z 569.994,A -85,B 0,C 180,E1 -18844.583,E2 -18844.583} C_VEL
LIN {X 0,Y 256.28,Z 560.544,A -85,B 0,C 180,E1 -18845.976,E2 -18845.976} C_VEL
LIN {X 0,Y 253.903,Z 555.939,A -85,B 0,C 180,E1 -18846.708,E2 -18846.708} C_VEL
LIN {X 0,Y 252.235,Z 549.336,A -85,B 0,C 180,E1 -18849.854,E2 -18849.854} C_VEL
LIN {X 0,Y 250.476,Z 543.072,A -85,B 0,C 180,E1 -18853.152,E2 -18853.152} C_VEL
LIN {X 0,Y 249.032,Z 538.463,A -85,B 0,C 180,E1 -18855.966,E2 -18855.966} C_VEL
LIN {X 0,Y 249.028,Z 538.462,A -85,B 0,C 180,E1 -18859.638,E2 -18859.638} C_VEL
LIN {X 0,Y 249.067,Z 538.456,A -85,B 0,C 180,E1 -18863.66,E2 -18863.66} C_VEL
LIN {X 0,Y 249.038,Z 538.464,A -85,B 0,C 180,E1 -18867.844,E2 -18867.844} C_VEL
LIN {X 0,Y 249.094,Z 538.455,A -85,B 0,C 180,E1 -18871.337,E2 -18871.337} C_VEL
LIN {X 0,Y 249.148,Z 538.444,A -85,B 0,C 180,E1 -18874.967,E2 -18874.967} C_VEL
LIN {X 0,Y 249.107,Z 538.451,A -85,B 0,C 180,E1 -18880.21,E2 -18880.21} C_VEL
LIN {X 0,Y 249.238,Z 538.433,A -85,B 0,C 180,E1 -18883.621,E2 -18883.621} C_VEL
LIN {X 0,Y 249.248,Z 538.439,A -85,B 0,C 180,E1 -18888.616,E2 -18888.616} C_VEL
LIN {X 0,Y 249.475,Z 538.409,A -85,B 0,C 180,E1 -18891.902,E2 -18891.902} C_VEL
LIN {X 0,Y 249.432,Z 538.408,A -85,B 0,C 180,E1 -18896.769,E2 -18896.769} C_VEL
LIN {X 0,Y 249.73,Z 538.372,A -85,B 0,C 180,E1 -18899.999,E2 -18899.999} C_VEL
LIN {X 0,Y 249.435,Z 538.409,A -85,B 0,C 180,E1 -18903.23,E2 -18903.23} C_VEL
LIN {X 0,Y 249.437,Z 538.408,A -85,B 0,C 180,E1 -18906.704,E2 -18906.704} C_VEL
LIN {X 0,Y 249.338,Z 538.425,A -85,B 0,C 180,E1 -18909.736,E2 -18909.736} C_VEL
LIN {X 0,Y 249.232,Z 538.59,A -85,B 0,C 180,E1 -18914.336,E2 -18914.336} C_VEL
LIN {X 0,Y 250.189,Z 541.274,A -85,B 0,C 180,E1 -18914.695,E2 -18914.695} C_VEL
LIN {X 0,Y 252.419,Z 543.725,A -85,B 0,C 180,E1 -18915.337,E2 -18915.337} C_VEL
LIN {X 0,Y 254.538,Z 547.179,A -85,B 0,C 180,E1 -18915.976,E2 -18915.976} C_VEL
LIN {X 0,Y 260.575,Z 556.534,A -85,B 0,C 180,E1 -18917.663,E2 -18917.663} C_VEL
LIN {X 0,Y 266.307,Z 566.488,A -85,B 0,C 180,E1 -18919.174,E2 -18919.174} C_VEL
LIN {X 0,Y 271.783,Z 578.035,A -85,B 0,C 180,E1 -18920.579,E2 -18920.579} C_VEL
LIN {X 0,Y 272.819,Z 580.457,A -85,B 0,C 180,E1 -18920.843,E2 -18920.843} C_VEL
LIN {X 0,Y 269.697,Z 643.028,A -85,B 0,C 180,E1 -18922.72,E2 -18922.72} C_VEL
LIN {X 0,Y 268.481,Z 656.457,A -85,B 0,C 180,E1 -18923.42,E2 -18923.42} C_VEL
LIN {X 0,Y 267.001,Z 668.792,A -85,B 0,C 180,E1 -18924.374,E2 -18924.374} C_VEL
LIN {X 0,Y 265.032,Z 680.883,A -85,B 0,C 180,E1 -18925.634,E2 -18925.634} C_VEL
LIN {X 0,Y 262.731,Z 692.468,A -85,B 0,C 180,E1 -18927.191,E2 -18927.191} C_VEL
LIN {X 0,Y 260.347,Z 702.393,A -85,B 0,C 180,E1 -18928.877,E2 -18928.877} C_VEL
LIN {X 0,Y 257.746,Z 712.248,A -85,B 0,C 180,E1 -18931.004,E2 -18931.004} C_VEL
LIN {X 0,Y 255.363,Z 720.279,A -85,B 0,C 180,E1 -18933.17,E2 -18933.17} C_VEL
LIN {X 0,Y 253.097,Z 727.536,A -85,B 0,C 180,E1 -18935.67,E2 -18935.67} C_VEL
LIN {X 0,Y 251.068,Z 733.613,A -85,B 0,C 180,E1 -18938.393,E2 -18938.393} C_VEL
LIN {X 0,Y 249.795,Z 737.33,A -85,B 0,C 180,E1 -18940.569,E2 -18940.569} C_VEL
LIN {X 0,Y 248.844,Z 740.188,A -85,B 0,C 180,E1 -18942.753,E2 -18942.753} C_VEL
LIN {X 0,Y 248.015,Z 742.373,A -85,B 0,C 180,E1 -18945.106,E2 -18945.106} C_VEL
LIN {X 0,Y 247.4,Z 743.727,A -85,B 0,C 180,E1 -18947.61,E2 -18947.61} C_VEL
LIN {X 0,Y 247.017,Z 744.124,A -85,B 0,C 180,E1 -18950.19,E2 -18950.19} C_VEL
LIN {X 0,Y 246.929,Z 743.249,A -85,B 0,C 180,E1 -18953.296,E2 -18953.296} C_VEL
LIN {X 0,Y 247.092,Z 741.708,A -85,B 0,C 180,E1 -18955.571,E2 -18955.571} C_VEL
LIN {X 0,Y 247.607,Z 738.636,A -85,B 0,C 180,E1 -18958.375,E2 -18958.375} C_VEL
LIN {X 0,Y 248.395,Z 734.007,A -85,B 0,C 180,E1 -18961.293,E2 -18961.293} C_VEL
LIN {X 0,Y 249.322,Z 728.679,A -85,B 0,C 180,E1 -18963.807,E2 -18963.807} C_VEL
LIN {X 0,Y 250.628,Z 721.449,A -85,B 0,C 180,E1 -18966.448,E2 -18966.448} C_VEL
LIN {X 0,Y 252.083,Z 713.498,A -85,B 0,C 180,E1 -18968.751,E2 -18968.751} C_VEL
LIN {X 0,Y 253.673,Z 704.769,A -85,B 0,C 180,E1 -18970.793,E2 -18970.793} C_VEL
LIN {X 0,Y 255.374,Z 694.518,A -85,B 0,C 180,E1 -18972.717,E2 -18972.717} C_VEL
LIN {X 0,Y 257.009,Z 683.705,A -85,B 0,C 180,E1 -18974.334,E2 -18974.334} C_VEL
LIN {X 0,Y 258.58,Z 671.737,A -85,B 0,C 180,E1 -18975.741,E2 -18975.741} C_VEL
LIN {X 0,Y 259.817,Z 659.165,A -85,B 0,C 180,E1 -18976.85,E2 -18976.85} C_VEL
LIN {X 0,Y 260.743,Z 646.491,A -85,B 0,C 180,E1 -18977.651,E2 -18977.651} C_VEL
LIN {X 0,Y 261.364,Z 633.804,A -85,B 0,C 180,E1 -18978.162,E2 -18978.162} C_VEL
LIN {X 0,Y 263.664,Z 572.585,A -85,B 0,C 180,E1 -18979.933,E2 -18979.933} C_VEL
LIN {X 0,Y 259.15,Z 560.773,A -85,B 0,C 180,E1 -18980.755,E2 -18980.755} C_VEL
LIN {X 0,Y 249.586,Z 539.158,A -85,B 0,C 180,E1 -18982.492,E2 -18982.492} C_VEL
LIN {X 0,Y 249.448,Z 538.414,A -85,B 0,C 180,E1 -18982.615,E2 -18982.615} C_VEL
LIN {X 0,Y 249.674,Z 538.385,A -85,B 0,C 180,E1 -18988.387,E2 -18988.387} C_VEL
LIN {X 0,Y 249.674,Z 538.384,A -85,B 0,C 180,E1 -18991.613,E2 -18991.613} C_VEL
LIN {X 0,Y 249.459,Z 538.411,A -85,B 0,C 180,E1 -18996.47,E2 -18996.47} C_VEL
LIN {X 0,Y 249.422,Z 538.414,A -85,B 0,C 180,E1 -18999.733,E2 -18999.733} C_VEL
